(* PLC project SixAxisBoxPicker_Task.project, CODESYS CODESYS V3.5 SP16 Patch 4 for Safety V1.6.1 *)
(* stored: creationDateTime 2022-02-01T19:12:31.3073643, modificationDateTime 2022-02-01T19:06:40.3294124 *)

{attribute 'qualified_only'}
{attribute 'strict'}
{attribute 'to_string'}
TYPE
  E_mcMotionFbType :
  (
    moveCrcAbs := 0,
    moveCrcRel,
    moveDirAbs,
    moveDirRel,
    moveLinAbs,
    moveLinRel,
    // enums have to begin from zero and be sequential for this to work
    TotalNumberOfEnums
  );
END_TYPE

TYPE
  ST_haltParams :
  STRUCT
    lrDec     : LREAL;
    lrJrk     : LREAL;
    lrAccFctr : LREAL                         := 1;
    lrJrkFctr : LREAL                         := 1;
    smcCrdSys : SM3_Robotics.SMC_COORD_SYSTEM := SM3_Robotics.SMC_COORD_SYSTEM.ACS; // for logging halted position
  END_STRUCT
END_TYPE

TYPE
  ST_mcMoveParams :
  STRUCT
    eMcMotionFbType : E_mcMotionFbType;
    stMoveDirParams : ST_moveDirParams;
    stMoveCrcParams : ST_moveCrcParams;
    stMoveLinParams : ST_moveLinParams;
  END_STRUCT
END_TYPE

TYPE
  ST_moveCrcParams :
  STRUCT
    smcCrcMod       : SM3_Robotics.SMC_CIRC_MODE;
    smcPosRef_auxPt : SM3_Robotics.SMC_POS_REF;
    smcPosRef_endPt : SM3_Robotics.SMC_POS_REF;
    mcCrcPathChoice : SM3_Robotics.MC_CIRC_PATHCHOICE;
    lrVel           : LREAL;
    lrAcc           : LREAL;
    lrDec           : LREAL;
    lrJrk           : LREAL;
    smcCrdSys       : SM3_Robotics.SMC_COORD_SYSTEM;
    mcBufMode       : SM3_Common.MC_BUFFER_MODE       := SM3_Common.MC_BUFFER_MODE.Aborting;
    mcTrnMode       : SM3_Robotics.MC_TRANSITION_MODE := SM3_Robotics.MC_TRANSITION_MODE.TMNone;
    arrTrnPrm       : ARRAY[0..(SMC_RCNST.MAX_TRANS_PARAMS - 1)] OF LREAL;
    smcOrnMod       : SM3_Robotics.SMC_ORIENTATION_MODE;
    lrVelFctr       : LREAL := 1;
    lrAccFctr       : LREAL := 1;
    lrJrkFctr       : LREAL := 1;
  END_STRUCT
END_TYPE

TYPE
  ST_moveDirParams :
  STRUCT
    smcPosRef : SM3_Robotics.SMC_POS_REF;
    smcPtpTyp : SM3_Robotics.SMC_PTP_MOVEMENT_TYPE;
    smcCrdSys : SM3_Robotics.SMC_COORD_SYSTEM;
    mcBufMode : SM3_Common.MC_BUFFER_MODE       := SM3_Common.MC_BUFFER_MODE.Aborting;
    mcTrnMode : SM3_Robotics.MC_TRANSITION_MODE := SM3_Robotics.MC_TRANSITION_MODE.TMNone;
    arrTrnPrm : ARRAY[0..(SMC_RCNST.MAX_TRANS_PARAMS - 1)] OF LREAL;
    lrVelFctr : LREAL := 1;
    lrAccFctr : LREAL := 1;
    lrJrkFctr : LREAL := 1;
  END_STRUCT
END_TYPE

TYPE
  ST_moveLinParams :
  STRUCT
    smcPosRef : SM3_Robotics.SMC_POS_REF;
    lrVel     : LREAL;
    lrAcc     : LREAL;
    lrDec     : LREAL;
    lrJrk     : LREAL;
    smcCrdSys : SM3_Robotics.SMC_COORD_SYSTEM;
    mcBufMode : SM3_Common.MC_BUFFER_MODE       := SM3_Common.MC_BUFFER_MODE.Aborting;
    mcTrnMode : SM3_Robotics.MC_TRANSITION_MODE := SM3_Robotics.MC_TRANSITION_MODE.TMNone;
    arrTrnPrm : ARRAY[0..(SMC_RCNST.MAX_TRANS_PARAMS - 1)] OF LREAL;
    smcOrnMod : SM3_Robotics.SMC_ORIENTATION_MODE;
    lrVelFctr : LREAL := 1;
    lrAccFctr : LREAL := 1;
    lrJrkFctr : LREAL := 1;
  END_STRUCT
END_TYPE

TYPE
  ST_methConfig :
  STRUCT
    xGroupPowerOff : BOOL;
    xGroupPowerOn  : BOOL;
    xGroupEnable   : BOOL;
    xGroupDisable  : BOOL;
    xGroupHalt     : BOOL;
    xMoveCrcAbs    : BOOL;
    xMoveDirAbs    : BOOL;
    xCloseGripper  : BOOL;
    xOpenGripper   : BOOL;
  END_STRUCT
END_TYPE

TYPE
  T_MaxString : STRING(1000);
END_TYPE

(* global variable list GVL_Diag *)
VAR_GLOBAL
	
	//-------------------
	// EtherCAT diagnosis
	//-------------------
	ECDiag : FB_ECDiag;	// Instance of Ethercat Diagnosis

	MyECSlaves : stECSlaves := // Input Values for EtherCAT Diagnosis 		
		(
			uiNoSlaves := 10,
			arMyProductID := 
			[
			16#0002CF2F,	// FIO_Buskoppler_16DI_16DO	
			16#0002D7A8,  	// Safety PLC
			16#0002ECAD,  	// Kuhnke_FIO_Safety_SDI16_SDO4_1
			16#0002ECAD,  	// Kuhnke_FIO_Safety_SDI16_SDO4_2
			16#00000201, 	// Synapticon Somanet
			16#00000201, 	// Synapticon Somanet
			16#00000201, 	// Synapticon Somanet
			16#00000201, 	// Synapticon Somanet
			16#00000201, 	// Synapticon Somanet
			16#00000201 	// Synapticon Somanet
			]
		);	

	//-------------------
	// Motion diagnosis
	//-------------------
	AxisDiag : FB_AxisDiag;// Instance of Axis Diagnosis

	MyAxis : stAxis := 		// Input Values for Axis Diagnosis 
		(
		uiNoAxis := INT_TO_UINT(iNoConfigAxis),		// Number of Axis in project	
		arMyAxis :=			// Pointer to Axis 
			[
			ADR(A1),
			ADR(A2),
			ADR(A3),
			ADR(A4)
			]
		);
	
	//-------------------
	// Group diagnosis
	//-------------------
	GroupDiag : FB_GroupDiag;// Instance of Group Diagnosis

	//-------------------
	// Safety diagnosis
	//-------------------
	SafetyIODiag1 : FB_SafetyIODiag;// Instance of SafetyIO Diagnosis
	SafetyIODiag2 : FB_SafetyIODiag;// Instance of SafetyIO Diagnosis
	
	//-------------------
	// Task diagnosis
	//-------------------
	TaskDiag : FB_TaskDiag ; // Instance of Task Diagnosis
	MyTask : stTask := 		// Input Values for Task Diagnosis 
		(
			sAppName := 'Application',
			Watchdog :=
			[
				(Active := TRUE,WDTime:= 4000,Sensitivity:=2),  // Watchdog EtherCAT Task 1
				(Active := TRUE,WDTime:= 20000,Sensitivity:=2), // Watchdog Planning Task 2
				(Active := FALSE)								// Watchdog Settings Task 3
			]			
		);

END_VAR

INTERFACE I_machineState
METHOD METH_grpPwrOn
END_METHOD
METHOD METH_grpPwrOff
END_METHOD
METHOD METH_openGripper
END_METHOD
METHOD METH_groupHalt
VAR_INPUT
  stHaltParams : ST_haltParams;
END_VAR
VAR_OUTPUT
  xHaltFinished : BOOL;
END_VAR
END_METHOD
METHOD METH_closeGripper
END_METHOD
METHOD METH_moveToPosition
VAR_IN_OUT
  mcMoveLinkedList : COL.LinkedList;
END_VAR
VAR_OUTPUT
  xMotionFinished : BOOL;
END_VAR
END_METHOD
METHOD METH_groupEnable
END_METHOD
METHOD METH_groupDisable
END_METHOD
END_INTERFACE

INTERFACE I_mcMoveElement EXTENDS COL.IElement
METHOD METH_executeMcMove
VAR_IN_OUT
  axisGrpRefSm3 : SM3_Robotics.AXIS_GROUP_REF_SM3;
END_VAR
VAR_OUTPUT
  xDone        : BOOL;
  xBusy        : BOOL;
  xActive      : BOOL;
  xCmdAborted  : BOOL;
  xCmdAccepted : BOOL;
  xError       : BOOL;
  smcError     : SM3_Error.SMC_ERROR;
  smcMvmtId    : SM3_Common.SMC_Movement_Id;
END_VAR
END_METHOD
METHOD METH_resetMcMove
VAR_IN_OUT
  axisGrpRefSm3 : SM3_Robotics.AXIS_GROUP_REF_SM3;
END_VAR
END_METHOD
METHOD METH_setMcMoveParams
VAR_INPUT
  stMcMoveParams : ST_mcMoveParams;
  uliMotionIndx  : ULINT;
END_VAR
END_METHOD
PROPERTY INTERNAL PROP_mcMoveCrcAbs : SM3_Robotics.MC_MoveCircularAbsolute
END_PROPERTY
PROPERTY INTERNAL PROP_mcMoveCrcRel : SM3_Robotics.MC_MoveCircularRelative
END_PROPERTY
PROPERTY PROP_motionIndx : ULINT
END_PROPERTY
PROPERTY PROP_stMcMoveParams : ST_mcMoveParams
END_PROPERTY
PROPERTY INTERNAL PROP_mcMoveDirAbs : SM3_Robotics.MC_MoveDirectAbsolute
END_PROPERTY
PROPERTY INTERNAL PROP_mcMoveDirRel : SM3_Robotics.MC_MoveDirectRelative
END_PROPERTY
PROPERTY INTERNAL PROP_mcMoveLinAbs : SM3_Robotics.MC_MoveLinearAbsolute
END_PROPERTY
PROPERTY INTERNAL PROP_mcMoveLinRel : SM3_Robotics.MC_MoveLinearRelative
END_PROPERTY
END_INTERFACE

TYPE U_lrealToRawLintBits : UNION
  lrVal : LREAL;
  liVal : LINT;
END_UNION;
END_TYPE

FUNCTION F_getCommaDelimitedName : STRING
VAR_IN_OUT
  sCommaDelimitedNames : STRING; // comma delimited string
END_VAR
VAR
  sComma    : STRING := ',';
  iSplitPos : INT;

  fbLogAdd : FB_logAdd(pCmpName:=ADR(__POUNAME()));
END_VAR

            IF Standard.LEN(sCommaDelimitedNames) > 0 THEN
  // returns zero if comma not found
  iSplitPos := Standard.FIND(sCommaDelimitedNames, sComma);

  // copy string and set position to last character if comma not found
  IF iSplitPos = 0 THEN
    F_getCommaDelimitedName := sCommaDelimitedNames;
    iSplitPos := Standard.LEN(sCommaDelimitedNames);
  ELSE
    // extract name without comma
    F_getCommaDelimitedName := Standard.LEFT(sCommaDelimitedNames, (iSplitPos - 1));
  END_IF

  // delete name including comma
  sCommaDelimitedNames := Standard.DELETE(sCommaDelimitedNames, iSplitPos, 1);
ELSE
  fbLogAdd.METH_appendLog('Axis names string empty! Was it comma delimited? Were there too few axis names?');
  fbLogAdd.METH_printAppendedLogs();
  F_getCommaDelimitedName := '$00';
END_IF

          
END_FUNCTION

FUNCTION_BLOCK FB_logAdd
VAR
  sCmpName : STRING;
  sCurrLog : T_MaxString;

  // to check for duplicate states or log messages
  sPrevName : STRING      := '$00';
  sPrevLog  : T_MaxString := '$00';

  // for use as delimiter
  sNewline : STRING := '$0A';

  // does not need to be set beforehand as only used internally
  udiInternalCmpId : UDINT;
END_VAR

            
          

METHOD METH_appendLog
VAR_INPUT
  sLog     : T_MaxString;
  xNewline : BOOL := FALSE;
END_VAR
VAR
  sErrLog : STRING;
END_VAR
                  TM.Stu.StrConcatA(pstFrom:=ADR(sLog),
                  pstTo:=ADR(sCurrLog),
                  iBufferSize:=UINT_TO_INT(SIZEOF(sCurrLog)));

IF xNewline THEN
  TM.Stu.StrConcatA(pstFrom:=ADR(sNewline),
                    pstTo:=ADR(sCurrLog),
                    iBufferSize:=UINT_TO_INT(SIZEOF(sCurrLog)));
END_IF

IF TM.Stu.StrLenA(ADR(sCurrLog)) = (SIZEOF(sCurrLog) - 1) THEN
  sErrLog := Standard.CONCAT('SIZEOF(sCurrLog) = ', UINT_TO_STRING(SIZEOF(sCurrLog)));
  sErrLog := Standard.CONCAT(sErrLog, ' but it is not large enough for logger!');

  METH_printError(sErrLog);
END_IF

                
END_METHOD

METHOD METH_printAppendedLogs
VAR_INPUT
  sCmpName      : STRING := '$00';
  udiCmpVer     : UDINT  := 16#1;
  udiLogClass   : UDINT  := SM3_Basic.CmpLog.LogClass.LOG_USER_NOTIFY;
  udiErrorClass : UDINT  := SM3_Basic.Errors.ERR_FAILED;
END_VAR
VAR
  iSplitPos : INT         := 0;
  sSplitLog : STRING(255) := '$00';
END_VAR
                  // use persistent variable if not provided otherwise replace persistent one
IF sCmpName = '$00' THEN
  sCmpName := THIS^.sCmpName;
ELSE
  THIS^.sCmpName := sCmpName;
END_IF

// print log only if either state (set to sCmpName) or log message is different
// StrCmpA returns zero if strings are equal
IF TM.Stu.StrCmpA(ADR(sPrevLog), ADR(sCurrLog)) <> 0 OR
   TM.Stu.StrCmpA(ADR(sPrevName), ADR(sCmpName)) <> 0 THEN

  // store component name and log content to prevent lots of duplicates
  sPrevName := sCmpName;
  sPrevLog := sCurrLog;

  // set metadata i.e. component name, version etc.
  SM3_Basic.Component_Manager.CMAddComponent2(pszComponent:=sCmpName,
                                              udiVersion:=udiCmpVer,
                                              udiCmpId:=ADR(udiInternalCmpId),
                                              pResult:=0);

  SM3_Basic.CmpLog.LogAdd2(hLogger:=SM3_Basic.CmpLog.LOG_STD_LOGGER,
                           udiCmpID:=udiInternalCmpId,
                           udiClassID:=udiLogClass,
                           udiErrorID:=udiErrorClass,
                           udiInfoID:=1,
                           pszInfo:='(*--------------------------------------------------*)');

  // limit for pszComponent is 29 chars (will become *** if longer)
  IF Standard.LEN(sCmpName) > 29 THEN
    // so print sCmpName before actual log
    sCmpName := Standard.CONCAT('Cmp=', sCmpName);
    SM3_Basic.CmpLog.LogAdd2(hLogger:=SM3_Basic.CmpLog.LOG_STD_LOGGER,
                             udiCmpID:=udiInternalCmpId,
                             udiClassID:=udiLogClass,
                             udiErrorID:=udiErrorClass,
                             udiInfoID:=1,
                             pszInfo:=sCmpName);
  END_IF

  // split string using newline as delimiter
  WHILE TM.Stu.StrLenA(ADR(sCurrLog)) > 0 DO
    // StrFindA returns zero if substring at pst2 not found
    iSplitPos := TM.Stu.StrFindA(pst1:=ADR(sCurrLog),
                                 pst2:=ADR(sNewline),
                                 uiSearchStart:=1);

    // copy string and set position to last character if newline not found
    IF iSplitPos = 0 THEN
      sSplitLog := sCurrLog;
      iSplitPos := DINT_TO_INT(TM.Stu.StrLenA(ADR(sCurrLog)));
    ELSE
      // extract string without newline
      TM.Stu.StrMidA(pst:=ADR(sCurrLog),
                     uiInputBufferSize:=SIZEOF(sCurrLog),
                     iLength:=(iSplitPos - 1), // do not include newline
                     iPosition:=1,
                     pstResult:=ADR(sSplitLog),
                     uiResultBufferSize:=SIZEOF(sSplitLog));
    END_IF

    // delete extracted string and its corresponding newline from original
    TM.Stu.StrDeleteA(pby:=ADR(sCurrLog),
                      iLength:=iSplitPos, // include newline
                      iPosition:=1);

    // print extracted string with logger
    SM3_Basic.CmpLog.LogAdd2(hLogger:=SM3_Basic.CmpLog.LOG_STD_LOGGER,
                             udiCmpID:=udiInternalCmpId,
                             udiClassID:=udiLogClass,
                             udiErrorID:=udiErrorClass,
                             udiInfoID:=1,
                             pszInfo:=sSplitLog);
  END_WHILE
END_IF

// printing should flush buffer so delete anything remaining
TM.Stu.StrDeleteA(pby:=ADR(sCurrLog),
                  iLength:=DINT_TO_INT(TM.Stu.StrLenA(ADR(sCurrLog))),
                  iPosition:=1);

                
END_METHOD

//FB_Init is always available implicitly and it is used primarily for initialization.
//The return value is not evaluated. For a specific influence, you can also declare the
//methods explicitly and provide additional code there with the standard initialization
//code. You can evaluate the return value.
METHOD FB_Init : BOOL
VAR_INPUT
  bInitRetains : BOOL; // TRUE: the retain variables are initialized (reset warm / reset cold)
  bInCopyCode  : BOOL; // TRUE: the instance will be copied to the copy code afterward (online change) 
  pCmpName     : POINTER TO STRING;
END_VAR
                  // check if pointer is initialized before assigning
IF pCmpName <> 0 THEN
  THIS^.sCmpName := pCmpName^;
END_IF

                
END_METHOD

METHOD METH_appendTargetPositionLogs
VAR_INPUT
  smcCrdSys       : SM3_Robotics.SMC_COORD_SYSTEM;
  sAxisNames      : STRING; // comma delimited string
  smcPosRef       : SM3_Robotics.SMC_POS_REF;
  eMcMotionFbType : E_mcMotionFbType;
END_VAR
VAR
  diIndx : DINT;
END_VAR
                  IF smcCrdSys = SM3_Robotics.SMC_COORD_SYSTEM.ACS THEN
  METH_appendLog(sLog:='{');
  METH_appendLog(sLog:=sAxisNames);
  METH_appendLog(sLog:='}',
                 xNewline:=TRUE);
ELSE
  METH_appendLog(sLog:='{X,Y,Z,A,B,C}',
                 xNewline:=TRUE);
END_IF

METH_appendLog(sLog:='{');

FOR diIndx := LOWER_BOUND(smcPosRef.v, 1) TO UPPER_BOUND(smcPosRef.v, 1) BY 1 DO
  METH_appendLog(sLog:=LREAL_TO_STRING(smcPosRef.v[diIndx]));

  IF diIndx < UPPER_BOUND(smcPosRef.v, 1) THEN
    METH_appendLog(sLog:=',');
  END_IF
END_FOR

METH_appendLog(sLog:='}',
               xNewline:=TRUE);
							 
METH_appendLog(sLog:='with ');

METH_appendLog(sLog:=TO_STRING(eMcMotionFbType),
							 xNewline:=TRUE);

METH_appendLog(sLog:='in ');

CASE smcCrdSys OF
  SM3_Robotics.SMC_COORD_SYSTEM.ACS:
    METH_appendLog(sLog:='Axis Coordinate System',
                   xNewline:=TRUE);
  SM3_Robotics.SMC_COORD_SYSTEM.MCS:
    METH_appendLog(sLog:='Machine Coordinate System',
                   xNewline:=TRUE);
  SM3_Robotics.SMC_COORD_SYSTEM.PCS_1:
    METH_appendLog(sLog:='PCS_1',
                   xNewline:=TRUE);
  SM3_Robotics.SMC_COORD_SYSTEM.PCS_2:
    METH_appendLog(sLog:='PCS_2',
                   xNewline:=TRUE);
  SM3_Robotics.SMC_COORD_SYSTEM.TCS:
    METH_appendLog(sLog:='Tool Coordinate System',
                   xNewline:=TRUE);
  SM3_Robotics.SMC_COORD_SYSTEM.WCS:
    METH_appendLog(sLog:='World Coordinate System',
                   xNewline:=TRUE);
END_CASE

                
END_METHOD

METHOD METH_appendGrpStatusLog
VAR_IN_OUT
  axisGrpRefSm3 : SM3_Robotics.AXIS_GROUP_REF_SM3;
END_VAR
VAR_INPUT
  sGrpName : STRING;
END_VAR
VAR
  mcGrpReadStatus : SM3_Robotics.MC_GroupReadStatus;
END_VAR
                  mcGrpReadStatus(AxisGroup:=axisGrpRefSm3, Enable:=TRUE);

IF mcGrpReadStatus.Error THEN
  METH_printError(SM3_Error.SMC_ErrorString(ErrorID:=mcGrpReadStatus.ErrorID,
                                            Language:=SM3_Error.SMC_LANGUAGE_TYPE.english));

  RETURN;
END_IF

IF mcGrpReadStatus.Valid THEN
  METH_appendLog('Axis: ');
  METH_appendLog(sGrpName);
  METH_appendLog(' Status: ');

  IF mcGrpReadStatus.GroupDisabled THEN
    METH_appendLog('disabled');
  ELSIF mcGrpReadStatus.GroupStandby THEN
    METH_appendLog('standby');
  ELSIF mcGrpReadStatus.GroupMoving THEN
    METH_appendLog('moving');
  ELSIF mcGrpReadStatus.GroupHoming THEN
    METH_appendLog('homing');
  ELSIF mcGrpReadStatus.GroupStopping THEN
    METH_appendLog('stopping');
  ELSIF mcGrpReadStatus.GroupErrorStop THEN
    METH_appendLog('errorstop');
  END_IF

  // remember to add newline as used as delimiter by logger
  METH_appendLog(sNewline);
END_IF

                
END_METHOD

METHOD PRIVATE METH_printError
VAR_INPUT
  sErrLog : STRING;
END_VAR
VAR
  sTempLog  : T_MaxString;
  sTempName : STRING;
END_VAR
                  sTempLog := sCurrLog;
sTempName := sPrevName;

sCurrLog := sErrLog;
METH_printAppendedLogs(sCmpName:=__POUNAME());

sPrevName := sTempName;
sCurrLog := sTempLog;

                
END_METHOD

METHOD METH_appendStatusLogs
VAR_IN_OUT
  axisGrpRefSm3 : SM3_Robotics.AXIS_GROUP_REF_SM3;
END_VAR
VAR_INPUT
  sGrpName   : STRING;
  sAxisNames : STRING; // comma delimited string
END_VAR
VAR
  diIndx          : DINT;
  pAxisRefSm3     : POINTER TO SM3_Robotics.AXIS_REF_SM3;
END_VAR
                  IF axisGrpRefSm3.m_nNumAxes = 0 THEN
  METH_printError(Standard.CONCAT(sGrpName, ' has no axes!'));
  RETURN;
END_IF

FOR diIndx := LOWER_BOUND(axisGrpRefSm3.m_aAxes, 1) TO UPPER_BOUND(axisGrpRefSm3.m_aAxes, 1) BY 1 DO
  pAxisRefSm3 := axisGrpRefSm3.m_aAxes[diIndx].GetAxisRefPointer();
  METH_appendAxisStatusLog(axisRefSm3:=pAxisRefSm3^,
                           sAxisName:=F_getCommaDelimitedName(sAxisNames));
END_FOR

METH_appendGrpStatusLog(axisGrpRefSm3:=axisGrpRefSm3,
                        sGrpName:=sGrpName);

                
END_METHOD

METHOD METH_appendAxisStatusLog
VAR_IN_OUT
  axisRefSm3 : SM3_Basic.AXIS_REF_SM3;
END_VAR
VAR_INPUT
  sAxisName : STRING;
END_VAR
VAR
  mcReadStatus : SM3_Basic.MC_ReadStatus;
  mcReadActPos : SM3_Basic.MC_ReadActualPosition;
END_VAR
                  mcReadStatus(Axis:=axisRefSm3, Enable:=TRUE);

IF mcReadStatus.Error THEN
  METH_printError(SM3_Error.SMC_ErrorString(ErrorID:=mcReadStatus.ErrorID,
                                            Language:=SM3_Error.SMC_LANGUAGE_TYPE.english));

  RETURN;
END_IF

IF mcReadStatus.Valid THEN
  METH_appendLog('Axis: ');
  METH_appendLog(sAxisName);
  METH_appendLog(' Status: ');

  IF mcReadStatus.Disabled THEN
    METH_appendLog('disabled');
  ELSIF mcReadStatus.Errorstop THEN
    METH_appendLog('errorstop');
  ELSIF mcReadStatus.Stopping THEN
    METH_appendLog('stopping');
  ELSIF mcReadStatus.StandStill THEN
    METH_appendLog('standstill');
  ELSIF mcReadStatus.DiscreteMotion THEN
    METH_appendLog('discrete_motion');
  ELSIF mcReadStatus.ContinuousMotion THEN
    METH_appendLog('continuous_motion');
  ELSIF mcReadStatus.SynchronizedMotion THEN
    METH_appendLog('synchronized_motion');
  ELSIF mcReadStatus.Homing THEN
    METH_appendLog('homing');
  END_IF

  IF mcReadStatus.ConstantVelocity THEN
    METH_appendLog(' Speed: ConstantVelocity');
  ELSIF mcReadStatus.Accelerating THEN
    METH_appendLog(' Speed: Accelerating');
  ELSIF mcReadStatus.Decelerating THEN
    METH_appendLog(' Speed: Decelerating');
  END_IF

END_IF

mcReadActPos(Axis:=axisRefSm3,
             Enable:=TRUE);

IF mcReadActPos.Error THEN
  // remember to add newline as used as delimiter by logger
  METH_appendLog(sNewline);

  METH_printError(SM3_Error.SMC_ErrorString(ErrorID:=mcReadActPos.ErrorID,
                                            Language:=SM3_Error.SMC_LANGUAGE_TYPE.english));

  RETURN;
END_IF

IF mcReadActPos.Valid THEN
  METH_appendLog(' Position: ');
  METH_appendLog(LREAL_TO_STRING(mcReadActPos.Position));
END_IF

// remember to add newline as used as delimiter by logger
METH_appendLog(sNewline);

                
END_METHOD

METHOD METH_appendCurrentPositionLogs
VAR_IN_OUT
  axisGrpRefSm3 : SM3_Robotics.AXIS_GROUP_REF_SM3;
END_VAR
VAR_INPUT
  smcCrdSys  : SM3_Robotics.SMC_COORD_SYSTEM;
  sAxisNames : STRING; // comma delimted string
END_VAR
VAR
  mcGrpReadActPos : SM3_Robotics.MC_GroupReadActualPosition;
  diIndx          : DINT;
  sIndividualName : STRING;
  sCoordNames     : STRING := 'X,Y,Z,A,B,C';
END_VAR
                  mcGrpReadActPos(AxisGroup:=axisGrpRefSm3,
                Enable:=TRUE,
                CoordSystem:=smcCrdSys);

IF mcGrpReadActPos.Error THEN
  METH_printError(SM3_Error.SMC_ErrorString(ErrorID:=mcGrpReadActPos.ErrorID,
                                            Language:=SM3_Error.SMC_LANGUAGE_TYPE.english));

  RETURN;
END_IF

IF mcGrpReadActPos.Valid THEN
  METH_appendLog(sLog:='Current position:',
                 xNewline:=TRUE);

  FOR diIndx := LOWER_BOUND(mcGrpReadActPos.Position.v, 1) TO UPPER_BOUND(mcGrpReadActPos.Position.v, 1) BY 1 DO

    IF diIndx = LOWER_BOUND(mcGrpReadActPos.Position.v, 1) THEN
      METH_appendLog(sLog:='{ ');
    ELSE
      METH_appendLog(sLog:='  '); // blank space for better log alignment
    END_IF

    IF smcCrdSys = SM3_Robotics.SMC_COORD_SYSTEM.ACS THEN
      sIndividualName := F_getCommaDelimitedName(sAxisNames);
    ELSE
      sIndividualName := F_getCommaDelimitedName(sCoordNames);
    END_IF

    METH_appendLog(sLog:=sIndividualName);
		METH_appendLog(sLog:=': ');
    METH_appendLog(sLog:=LREAL_TO_STRING(mcGrpReadActPos.Position.v[diIndx]));

    IF diIndx = UPPER_BOUND(mcGrpReadActPos.Position.v, 1) THEN
      METH_appendLog(sLog:=' }',
                     xNewline:=TRUE);
    ELSE
      METH_appendLog(sLog:=',',
                     xNewline:=TRUE);
    END_IF
  END_FOR

END_IF

                
END_METHOD
END_FUNCTION_BLOCK

FUNCTION_BLOCK INTERNAL ABSTRACT FB_abstractEndMachineState EXTENDS FB_abstractMachineState IMPLEMENTS I_machineState

            sStateFb := __POUNAME();

          

METHOD METH_groupEnable
                  IF stMethConfig.xGroupEnable THEN
  METH_appendStateFbLog();
  METH_appendStatusLogs();
  METH_appendInfoLog('Enabling axes...');
  METH_printInfo(__POUNAME());

  pFbMachine^.METH_setState(pFbMachine^.PROP_enablingAxesState);
END_IF

                
END_METHOD

METHOD METH_grpPwrOn
                  IF stMethConfig.xGroupPowerOn THEN
  METH_appendStateFbLog();
  METH_appendStatusLogs();
  METH_appendInfoLog('Powering on axes...');
  METH_printInfo(__POUNAME());

  pFbMachine^.METH_setState(pFbMachine^.PROP_poweringOnState);
END_IF

                
END_METHOD

METHOD METH_grpPwrOff
                  IF stMethConfig.xGroupPowerOff THEN
  METH_appendStateFbLog();
  METH_appendStatusLogs();
  METH_appendInfoLog('Powering off axes...');
  METH_printInfo(__POUNAME());

  pFbMachine^.METH_setState(pFbMachine^.PROP_poweringOffState);
END_IF

                
END_METHOD

METHOD METH_openGripper
                  // IF stMethConfig.xOpenGripper THEN
// 	
// END_IF                           
                
END_METHOD

METHOD METH_groupHalt
VAR_INPUT
  stHaltParams : ST_haltParams;
END_VAR
VAR_OUTPUT
  xHaltFinished : BOOL;
END_VAR
                  // default values cannot be set in abstract or interface method
xHaltFinished := FALSE;

IF stMethConfig.xGroupHalt THEN
  METH_appendStateFbLog();
  METH_appendStatusLogs();
  METH_appendInfoLog('Halting axes...');
  METH_printInfo(__POUNAME());

  pFbMachine^.METH_setState(pFbMachine^.PROP_haltingState);
END_IF

                
END_METHOD

METHOD METH_closeGripper
                  // IF stMethConfig.xCloseGripper THEN
// END_IF                           
                
END_METHOD

METHOD METH_moveToPosition
VAR_IN_OUT
  mcMoveLinkedList : COL.LinkedList;
END_VAR
VAR_OUTPUT
  xMotionFinished : BOOL;
END_VAR
VAR
  linkedListIterator : COL.LinkedListIterator;
  itfLinkedListElem  : COL.IElement;
  itfMcMoveElement   : I_mcMoveElement;
  stMcMoveParams     : ST_mcMoveParams;

  mcMoveLinkedListInfo  : __SYSTEM.VAR_INFO;
  itfLinkedListElemInfo : __SYSTEM.VAR_INFO;
  itfMcMoveElementInfo  : __SYSTEM.VAR_INFO;
END_VAR
                  // default values cannot be set in abstract or interface method
xMotionFinished := FALSE;

IF stMethConfig.xMoveDirAbs THEN

  mcMoveLinkedListInfo := __VARINFO(mcMoveLinkedList);

  IF mcMoveLinkedList.CountElements() <= 0 THEN
    METH_appendInfoLog('No elements in ');
    METH_appendInfoLog(mcMoveLinkedListInfo.Symbol);
    METH_appendInfoLog('!');
  ELSE
    mcMoveLinkedList.ElementIterator(itfIterator:=linkedListIterator);

    WHILE linkedListIterator.HasNext() DO
      linkedListIterator.Next(itfElement=>itfLinkedListElem);

      itfLinkedListElemInfo := __VARINFO(itfLinkedListElem);
      itfMcMoveElementInfo := __VARINFO(itfMcMoveElement);

      IF NOT __QUERYINTERFACE(itfLinkedListElem, itfMcMoveElement) THEN
        METH_appendInfoLog('Unable to convert ');
        METH_appendInfoLog(itfLinkedListElemInfo.Symbol);
        METH_appendInfoLog(' to ');
        METH_appendInfoLog(itfMcMoveElementInfo.Symbol);
        METH_appendInfoLog('!');
      ELSE
        METH_appendStateFbLog();
        METH_appendStatusLogs();
        METH_appendInfoLog('Moving to position...');

        stMcMoveParams := itfMcMoveElement.PROP_stMcMoveParams;

        CASE stMcMoveParams.eMcMotionFbType OF

          E_mcMotionFbType.moveCrcAbs:
            METH_appendInfoLog('Not implemented yet!');

          E_mcMotionFbType.moveCrcRel:
            METH_appendInfoLog('Not implemented yet!');

          E_mcMotionFbType.moveDirAbs:
            METH_appendTargetPositionLogs(smcCrdSys:=stMcMoveParams.stMoveDirParams.smcCrdSys,
                                          smcPosRef:=stMcMoveParams.stMoveDirParams.smcPosRef,
                                          eMcMotionFbType:=stMcMoveParams.eMcMotionFbType);

          E_mcMotionFbType.moveDirRel:
            METH_appendTargetPositionLogs(smcCrdSys:=stMcMoveParams.stMoveDirParams.smcCrdSys,
                                          smcPosRef:=stMcMoveParams.stMoveDirParams.smcPosRef,
                                          eMcMotionFbType:=stMcMoveParams.eMcMotionFbType);

          E_mcMotionFbType.moveLinAbs:
            METH_appendTargetPositionLogs(smcCrdSys:=stMcMoveParams.stMoveLinParams.smcCrdSys,
                                          smcPosRef:=stMcMoveParams.stMoveLinParams.smcPosRef,
                                          eMcMotionFbType:=stMcMoveParams.eMcMotionFbType);

          E_mcMotionFbType.moveLinRel:
            METH_appendTargetPositionLogs(smcCrdSys:=stMcMoveParams.stMoveLinParams.smcCrdSys,
                                          smcPosRef:=stMcMoveParams.stMoveLinParams.smcPosRef,
                                          eMcMotionFbType:=stMcMoveParams.eMcMotionFbType);

        END_CASE

        METH_printInfo(__POUNAME());
      END_IF
    END_WHILE
  END_IF

  pFbMachine^.METH_setState(pFbMachine^.PROP_movingToPositionState);
END_IF

                
END_METHOD

METHOD METH_groupDisable
                  IF stMethConfig.xGroupDisable THEN
  METH_appendStateFbLog();
  METH_appendStatusLogs();
  METH_appendInfoLog('Disabling axes...');
  METH_printInfo(__POUNAME());

  pFbMachine^.METH_setState(pFbMachine^.PROP_disablingAxesState);
END_IF

                
END_METHOD
END_FUNCTION_BLOCK

FUNCTION_BLOCK INTERNAL FB_disabledAxesState EXTENDS FB_abstractEndMachineState

            sStateFb := __POUNAME();

stMethConfig.xGroupPowerOff := TRUE;
stMethConfig.xGroupPowerOn  := FALSE;
stMethConfig.xGroupEnable   := TRUE;
stMethConfig.xGroupDisable  := FALSE;
stMethConfig.xMoveDirAbs    := FALSE;
stMethConfig.xGroupHalt     := FALSE;
stMethConfig.xCloseGripper  := FALSE;
stMethConfig.xOpenGripper   := FALSE;

          
END_FUNCTION_BLOCK

FUNCTION_BLOCK INTERNAL FB_enabledAxesState EXTENDS FB_abstractEndMachineState

            sStateFb := __POUNAME();

stMethConfig.xGroupPowerOff := FALSE;
stMethConfig.xGroupPowerOn  := FALSE;
stMethConfig.xGroupEnable   := FALSE;
stMethConfig.xGroupDisable  := TRUE;
stMethConfig.xMoveDirAbs    := TRUE;
stMethConfig.xGroupHalt     := TRUE;
stMethConfig.xCloseGripper  := TRUE;
stMethConfig.xOpenGripper   := TRUE;

          
END_FUNCTION_BLOCK

FUNCTION_BLOCK INTERNAL FB_haltedState EXTENDS FB_abstractEndMachineState

            sStateFb := __POUNAME();

stMethConfig.xGroupPowerOff := FALSE;
stMethConfig.xGroupPowerOn  := FALSE;
stMethConfig.xGroupEnable   := FALSE;
stMethConfig.xGroupDisable  := TRUE;
stMethConfig.xMoveDirAbs    := TRUE;
stMethConfig.xGroupHalt     := TRUE;
stMethConfig.xCloseGripper  := TRUE;
stMethConfig.xOpenGripper   := TRUE;

          
END_FUNCTION_BLOCK

FUNCTION_BLOCK INTERNAL FB_movedToPositionState EXTENDS FB_abstractEndMachineState

            sStateFb := __POUNAME();

stMethConfig.xGroupPowerOff := FALSE;
stMethConfig.xGroupPowerOn  := FALSE;
stMethConfig.xGroupEnable   := FALSE;
stMethConfig.xGroupDisable  := TRUE;
stMethConfig.xMoveDirAbs    := TRUE;
stMethConfig.xGroupHalt     := TRUE;
stMethConfig.xCloseGripper  := TRUE;
stMethConfig.xOpenGripper   := TRUE;

          
END_FUNCTION_BLOCK

FUNCTION_BLOCK INTERNAL FB_poweredOffState EXTENDS FB_abstractEndMachineState

            sStateFb := __POUNAME();

stMethConfig.xGroupPowerOff := FALSE;
stMethConfig.xGroupPowerOn  := TRUE;
stMethConfig.xGroupEnable   := FALSE;
stMethConfig.xGroupDisable  := FALSE;
stMethConfig.xMoveDirAbs    := FALSE;
stMethConfig.xGroupHalt     := FALSE;
stMethConfig.xCloseGripper  := FALSE;
stMethConfig.xOpenGripper   := FALSE;

          
END_FUNCTION_BLOCK

FUNCTION_BLOCK INTERNAL FB_poweredOnState EXTENDS FB_abstractEndMachineState

            sStateFb := __POUNAME();

stMethConfig.xGroupPowerOff := TRUE;
stMethConfig.xGroupPowerOn  := FALSE;
stMethConfig.xGroupEnable   := TRUE;
stMethConfig.xGroupDisable  := FALSE;
stMethConfig.xMoveDirAbs    := FALSE;
stMethConfig.xGroupHalt     := FALSE;
stMethConfig.xCloseGripper  := FALSE;
stMethConfig.xOpenGripper   := FALSE;

          
END_FUNCTION_BLOCK

FUNCTION_BLOCK INTERNAL ABSTRACT FB_abstractMachineState
VAR
  pFbMachine   : POINTER TO FB_machine;
  pFbLogAdd    : POINTER TO FB_logAdd; // centralized in FB_machine
  sStateFb     : STRING;
  stMethConfig : ST_methConfig;
END_VAR

            sStateFb := __POUNAME();

          

//FB_Init is always available implicitly and it is used primarily for initialization.
//The return value is not evaluated. For a specific influence, you can also declare the
//methods explicitly and provide additional code there with the standard initialization
//code. You can evaluate the return value.
METHOD FB_Init : BOOL
VAR_INPUT
  bInitRetains : BOOL; // TRUE: the retain variables are initialized (reset warm / reset cold)
  bInCopyCode  : BOOL; // TRUE: the instance will be copied to the copy code afterward (online change)   
  pFbMachine   : POINTER TO FB_machine;
END_VAR
                  THIS^.pFbMachine := pFbMachine;
THIS^.pFbLogAdd := THIS^.pFbMachine^.PROP_fbLogAddPointer;

                
END_METHOD

METHOD PROTECTED METH_printInfo
VAR_INPUT
  sCmpName : STRING;
END_VAR
                  pFbLogAdd^.METH_printAppendedLogs(sCmpName:=sCmpName,
                                  udiErrorClass:=SM3_Basic.CmpLog.LogClass.LOG_INFO);

                
END_METHOD

METHOD PROTECTED METH_printSmcError
VAR_INPUT
  smcErrorId : SM3_Error.SMC_ERROR;
  sCmpName   : STRING;
END_VAR
                  pFbLogAdd^.METH_appendLog(sLog:=SM3_Error.SMC_ErrorString(ErrorID:=smcErrorId,
                                                          Language:=SM3_Error.SMC_LANGUAGE_TYPE.english));

pFbLogAdd^.METH_printAppendedLogs(sCmpName:=sCmpName);

                
END_METHOD

METHOD PROTECTED METH_appendStatusLogs
                  pFbLogAdd^.METH_appendStatusLogs(axisGrpRefSm3:=pFbMachine^.PROP_axisGroupPointer^,
                                 sGrpName:=pFbMachine^.sGrpName,
                                 sAxisNames:=pFbMachine^.sAxisNames);

                
END_METHOD

METHOD PROTECTED METH_appendInfoLog
VAR_INPUT
  sInfoMsg : STRING;
END_VAR
                  pFbLogAdd^.METH_appendLog(sLog:=sInfoMsg,
                          xNewline:=TRUE);

                
END_METHOD

METHOD PROTECTED METH_appendTargetPositionLogs
VAR_INPUT
  smcCrdSys : SM3_Robotics.SMC_COORD_SYSTEM;
  smcPosRef : SM3_Robotics.SMC_POS_REF;
	eMcMotionFbType : E_mcMotionFbType;
END_VAR
                  pFbLogAdd^.METH_appendTargetPositionLogs(smcCrdSys:=smcCrdSys,
                                         sAxisNames:=pFbMachine^.sAxisNames,
                                         smcPosRef:=smcPosRef,
                                         eMcMotionFbType:=eMcMotionFbType);

                
END_METHOD

METHOD PROTECTED METH_appendStateFbLog
                  pFbLogAdd^.METH_appendLog(sLog:='Current state: ');
pFbLogAdd^.METH_appendLog(sLog:=sStateFb,
                          xNewline:=TRUE);

                
END_METHOD

METHOD PROTECTED METH_appendCurrentPositionLogs
VAR_INPUT
  smcCrdSys : SM3_Robotics.SMC_COORD_SYSTEM;
END_VAR
                  pFbLogAdd^.METH_appendCurrentPositionLogs(axisGrpRefSm3:=pFbMachine^.PROP_axisGroupPointer^,
                                          sAxisNames:=pFbMachine^.sAxisNames,
                                          smcCrdSys:=smcCrdSys);

                
END_METHOD
END_FUNCTION_BLOCK

FUNCTION_BLOCK FB_machine
VAR
  // everything initialized in FB_Init
  rAxisGrpRefSm3 : REFERENCE TO SM3_Robotics.AXIS_GROUP_REF_SM3;
  sGrpName       : STRING;
  sAxisNames     : STRING; // comma delimited string

  // logger used by FB_baseMachineState
  fbLogAdd : FB_logAdd(pCmpName:=ADR(__POUNAME()));

  // state pattern
  itfMachineState : I_machineState := fbPoweredOff;

  // end states
  fbPoweredOff      : FB_poweredOffState(THIS);
  fbPoweredOn       : FB_poweredOnState(THIS);
  fbEnabledAxes     : FB_enabledAxesState(THIS);
  fbDisabledAxes    : FB_disabledAxesState(THIS);
  fbHalted          : FB_haltedState(THIS);
  fbMovedToPosition : FB_movedToPositionState(THIS);
  // interim states
  fbPoweringOff      : FB_poweringOffState(THIS);
  fbPoweringOn       : FB_poweringOnState(THIS);
  fbEnablingAxes     : FB_enablingAxesState(THIS);
  fbDisablingAxes    : FB_disablingAxesState(THIS);
  fbHalting          : FB_haltingState(THIS);
  fbMovingToPosition : FB_movingToPositionState(THIS);
END_VAR

            
          

METHOD INTERNAL METH_setState
VAR_INPUT
  itfNewState : I_machineState;
END_VAR
                  itfMachineState := itfNewState;

                
END_METHOD

METHOD METH_groupEnable
                  itfMachineState.METH_groupEnable();

                
END_METHOD

//FB_Init is always available implicitly and it is used primarily for initialization.
//The return value is not evaluated. For a specific influence, you can also declare the
//methods explicitly and provide additional code there with the standard initialization
//code. You can evaluate the return value.
METHOD FB_Init : BOOL
VAR_INPUT
  bInitRetains   : BOOL; // TRUE: the retain variables are initialized (reset warm / reset cold)
  bInCopyCode    : BOOL; // TRUE: the instance will be copied to the copy code afterward (online change)
  rAxisGrpRefSm3 : REFERENCE TO SM3_Robotics.AXIS_GROUP_REF_SM3;
  sGrpName       : STRING;
  sAxisNames     : STRING; // comma delimited string
END_VAR
                  IF __ISVALIDREF(rAxisGrpRefSm3) THEN
	THIS^.rAxisGrpRefSm3 REF= rAxisGrpRefSm3;
END_IF
THIS^.sGrpName := sGrpName;
THIS^.sAxisNames := sAxisNames;

// initialize respective ST_methConfig 
// end states
THIS^.fbPoweredOff();
THIS^.fbPoweredOn();
THIS^.fbEnabledAxes();
THIS^.fbDisabledAxes();
THIS^.fbHalted();
// THIS^.fbMovedCrcAbs();
THIS^.fbMovedToPosition();
// interim states
THIS^.fbPoweringOff();
THIS^.fbPoweringOn();
THIS^.fbEnablingAxes();
THIS^.fbDisablingAxes();
THIS^.fbHalting();
// THIS^.fbMovingCrcAbs();
THIS^.fbMovingToPosition();

                
END_METHOD

METHOD METH_groupDisable
                  itfMachineState.METH_groupDisable();

                
END_METHOD

METHOD METH_grpPwrOn
                  itfMachineState.METH_grpPwrOn();

                
END_METHOD

METHOD METH_grpPwrOff
                  itfMachineState.METH_grpPwrOff();

                
END_METHOD

METHOD METH_moveToPosition
VAR_IN_OUT
  mcMoveLinkedList : COL.LinkedList;
END_VAR
VAR_OUTPUT
  xMotionFinished : BOOL;
END_VAR
                  itfMachineState.METH_moveToPosition(mcMoveLinkedList,
                                    xMotionFinished=>xMotionFinished);

                
END_METHOD

METHOD METH_groupHalt
VAR_INPUT
  stHaltParams : ST_haltParams;
END_VAR
VAR_OUTPUT
  xHaltFinished : BOOL;
END_VAR
                  itfMachineState.METH_groupHalt(stHaltParams:=stHaltParams,
                          xHaltFinished=>xHaltFinished);

                
END_METHOD

PROPERTY INTERNAL PROP_poweringOnState : I_machineState
GET
                    PROP_poweringOnState := fbPoweringOn;

                  
END_GET
END_PROPERTY

PROPERTY INTERNAL PROP_poweredOnState : I_machineState
GET
                    PROP_poweredOnState := fbPoweredOn;

                  
END_GET
END_PROPERTY

PROPERTY INTERNAL PROP_poweredOffState : I_machineState
GET
                    PROP_poweredOffState := fbPoweredOff;

                  
END_GET
END_PROPERTY

PROPERTY INTERNAL PROP_fbLogAddPointer : POINTER TO FB_logAdd
GET
                    PROP_fbLogAddPointer := ADR(fbLogAdd);

                  
END_GET
END_PROPERTY

PROPERTY PROP_axisGroupPointer : POINTER TO AXIS_GROUP_REF_SM3
GET
                    PROP_axisGroupPointer := ADR(rAxisGrpRefSm3);

                  
END_GET
END_PROPERTY

PROPERTY INTERNAL PROP_poweringOffState : I_machineState
GET
                    PROP_poweringOffState := fbPoweringOff;

                  
END_GET
END_PROPERTY

PROPERTY INTERNAL PROP_enabledAxesState : I_machineState
GET
                    PROP_enabledAxesState := fbEnabledAxes;

                  
END_GET
END_PROPERTY

PROPERTY INTERNAL PROP_enablingAxesState : I_machineState
GET
                    PROP_enablingAxesState := fbEnablingAxes;

                  
END_GET
END_PROPERTY

PROPERTY INTERNAL PROP_disabledAxesState : I_machineState
GET
                    PROP_disabledAxesState := fbDisabledAxes;

                  
END_GET
END_PROPERTY

PROPERTY INTERNAL PROP_disablingAxesState : I_machineState
GET
                    PROP_disablingAxesState := fbDisablingAxes;

                  
END_GET
END_PROPERTY

PROPERTY INTERNAL PROP_movedToPositionState : I_machineState
GET
                    PROP_movedToPositionState := fbMovedToPosition;

                  
END_GET
END_PROPERTY

PROPERTY INTERNAL PROP_movingToPositionState : I_machineState
GET
                    PROP_movingToPositionState := fbMovingToPosition;

                  
END_GET
END_PROPERTY

PROPERTY INTERNAL PROP_haltingState : I_machineState
GET
                    PROP_haltingState := fbHalting;

                  
END_GET
END_PROPERTY

PROPERTY INTERNAL PROP_haltedState : I_machineState
GET
                    PROP_haltedState := fbHalted;

                  
END_GET
END_PROPERTY
END_FUNCTION_BLOCK

FUNCTION_BLOCK INTERNAL ABSTRACT FB_abstractInterimMachineState EXTENDS FB_abstractMachineState IMPLEMENTS I_machineState

            sStateFb := __POUNAME();

          

METHOD METH_groupEnable
VAR
  mcGrpEnable : SM3_Robotics.MC_GroupEnable;
END_VAR
                  IF stMethConfig.xGroupEnable THEN
  mcGrpEnable(AxisGroup:=pFbMachine^.PROP_axisGroupPointer^,
              Execute:=TRUE);

  IF mcGrpEnable.Error THEN
    METH_printSmcError(smcErrorId:=mcGrpEnable.ErrorID,
                    sCmpName:=__POUNAME());

    RETURN;
  END_IF

  METH_appendStateFbLog();
  METH_appendStatusLogs();

  IF mcGrpEnable.Done THEN
    METH_appendInfoLog('Enabled axes');

    pFbMachine^.METH_setState(pFbMachine^.PROP_enabledAxesState);
  ELSE
    pFbMachine^.METH_setState(pFbMachine^.PROP_enablingAxesState);
  END_IF

  METH_printInfo(__POUNAME());

END_IF

                
END_METHOD

METHOD METH_openGripper
                  // IF stMethConfig.xOpenGripper THEN
// 	
// END_IF                             
                
END_METHOD

METHOD METH_groupHalt
VAR_INPUT
  stHaltParams : ST_haltParams;
END_VAR
VAR_OUTPUT
  xHaltFinished : BOOL;
END_VAR
VAR
  mcGrpHalt    : SM3_Robotics.MC_GroupHalt;
END_VAR
                  // default values cannot be set in abstract or interface method
xHaltFinished := FALSE;

IF stMethConfig.xGroupHalt THEN

  mcGrpHalt(AxisGroup:=pFbMachine^.PROP_axisGroupPointer^,
            Execute:=TRUE,
            Deceleration:=stHaltParams.lrDec,
            Jerk:=stHaltParams.lrJrk,
            AccFactor:=stHaltParams.lrAccFctr,
            JerkFactor:=stHaltParams.lrJrkFctr);

  IF mcGrpHalt.Error THEN
    METH_printSmcError(smcErrorId:=mcGrpHalt.ErrorID,
                    sCmpName:=__POUNAME());

    RETURN;
  END_IF

  METH_appendStateFbLog();
  METH_appendStatusLogs();

  IF mcGrpHalt.Done THEN
    METH_appendInfoLog('Halted');

    // remember to reset execute since persistent FB otherwise will not move to next position when called
    mcGrpHalt(AxisGroup:=pFbMachine^.PROP_axisGroupPointer^,
              Execute:=FALSE);

    xHaltFinished := TRUE;

    pFbMachine^.METH_setState(pFbMachine^.PROP_haltedState);
  ELSE
    pFbMachine^.METH_setState(pFbMachine^.PROP_haltingState);
  END_IF

  // axis positions already printed in METH_appendStatusLogs()
  IF stHaltParams.smcCrdSys <> SM3_Robotics.SMC_COORD_SYSTEM.ACS THEN
    METH_appendCurrentPositionLogs(smcCrdSys:=stHaltParams.smcCrdSys);
  END_IF

  METH_printInfo(__POUNAME());

END_IF

                
END_METHOD

METHOD METH_grpPwrOff
VAR
  smcGrpPwr : SM3_Robotics.SMC_GroupPower;
END_VAR
                  IF stMethConfig.xGroupPowerOff THEN
  smcGrpPwr(AxisGroup:=pFbMachine^.PROP_axisGroupPointer^,
            Enable:=TRUE,
            bRegulatorOn:=FALSE,
            bDriveStart:=FALSE);

  IF smcGrpPwr.Error THEN
    METH_printSmcError(smcErrorId:=smcGrpPwr.ErrorID,
                    sCmpName:=__POUNAME());

    RETURN;
  END_IF

  METH_appendStateFbLog();
  METH_appendStatusLogs();

  IF smcGrpPwr.Status THEN
    METH_appendInfoLog('Powered off axes');

    pFbMachine^.METH_setState(pFbMachine^.PROP_poweredOffState);
  ELSE
    pFbMachine^.METH_setState(pfbmachine^.PROP_poweringOffState);
  END_IF

  METH_printInfo(__POUNAME());

END_IF

                
END_METHOD

METHOD METH_grpPwrOn
VAR
  smcGrpPwr : SM3_Robotics.SMC_GroupPower;
END_VAR
                  IF stMethConfig.xGroupPowerOn THEN
  smcGrpPwr(AxisGroup:=pFbMachine^.PROP_axisGroupPointer^,
            Enable:=TRUE,
            bRegulatorOn:=TRUE,
            bDriveStart:=TRUE);

  IF smcGrpPwr.Error THEN
    METH_printSmcError(smcErrorId:=smcGrpPwr.ErrorID,
                    sCmpName:=__POUNAME());

    RETURN;
  END_IF

  METH_appendStateFbLog();
  METH_appendStatusLogs();

  IF smcGrpPwr.Status THEN
    METH_appendInfoLog('Powered on axes');

    pFbMachine^.METH_setState(pFbMachine^.PROP_poweredOnState);
  ELSE
    pFbMachine^.METH_setState(pfbmachine^.PROP_poweringOnState);
  END_IF

  METH_printInfo(__POUNAME());

END_IF

                
END_METHOD

METHOD METH_closeGripper
                  // IF stMethConfig.xCloseGripper THEN
// 	
// END_IF                             
                
END_METHOD

METHOD METH_moveToPosition
VAR_IN_OUT
  mcMoveLinkedList : COL.LinkedList;
END_VAR
VAR_OUTPUT
  xMotionFinished : BOOL;
END_VAR
VAR
	linkedListIterator : COL.LinkedListIterator;
  itfLinkedListElem  : COL.IElement;
  itfMcMoveElement   : I_mcMoveElement;
  stMcMoveParams     : ST_mcMoveParams;

  mcMoveLinkedListInfo  : __SYSTEM.VAR_INFO;
  itfLinkedListElemInfo : __SYSTEM.VAR_INFO;
  itfMcMoveElementInfo  : __SYSTEM.VAR_INFO;

  xDone        : BOOL;
  xBusy        : BOOL;
  xActive      : BOOL;
  xCmdAborted  : BOOL;
  xCmdAccepted : BOOL;
  xError       : BOOL;
  smcError     : SM3_Error.SMC_ERROR;
  smcMvmtId    : SM3_Common.SMC_Movement_Id;
END_VAR
                  // default values cannot be set in abstract or interface method
xMotionFinished := FALSE;

IF stMethConfig.xMoveDirAbs THEN

  mcMoveLinkedListInfo := __VARINFO(mcMoveLinkedList);

  IF mcMoveLinkedList.CountElements() <= 0 THEN
    METH_appendInfoLog('No elements in ');
    METH_appendInfoLog(mcMoveLinkedListInfo.Symbol);
    METH_appendInfoLog('!');
  ELSE
    mcMoveLinkedList.ElementIterator(itfIterator:=linkedListIterator);

    WHILE linkedListIterator.HasNext() DO
      linkedListIterator.Next(itfElement=>itfLinkedListElem);

      itfLinkedListElemInfo := __VARINFO(itfLinkedListElem);
      itfMcMoveElementInfo := __VARINFO(itfMcMoveElement);

      IF NOT __QUERYINTERFACE(itfLinkedListElem, itfMcMoveElement) THEN
        METH_appendInfoLog('Unable to convert ');
        METH_appendInfoLog(itfLinkedListElemInfo.Symbol);
        METH_appendInfoLog(' to ');
        METH_appendInfoLog(itfMcMoveElementInfo.Symbol);
        METH_appendInfoLog('!');
      ELSE
        itfMcMoveElement.METH_executeMcMove(axisGrpRefSm3:=pFbMachine^.PROP_axisGroupPointer^,
                                            xDone=>xDone,
                                            xBusy=>xBusy,
                                            xActive=>xActive,
                                            xCmdAborted=>xCmdAborted,
                                            xCmdAccepted=>xCmdAccepted,
                                            xError=>xError,
                                            smcError=>smcError,
                                            smcMvmtId=>smcMvmtId);

        IF xError THEN
          METH_printSmcError(smcErrorId:=smcError,
                             sCmpName:=__POUNAME());

          RETURN;
        END_IF

        METH_appendStateFbLog();
        METH_appendStatusLogs();

        stMcMoveParams := itfMcMoveElement.PROP_stMcMoveParams;

        IF xDone THEN
          METH_appendInfoLog('Moved to position');

          // need to implement method containing case statement for appendTargetPositionLogs
          METH_appendTargetPositionLogs(smcCrdSys:=stMcMoveParams.stMoveDirParams.smcCrdSys,
                                        smcPosRef:=stMcMoveParams.stMoveDirParams.smcPosRef,
                                        eMcMotionFbType:=E_mcMotionFbType.moveDirAbs);

          // remember to reset execute since persistent FB otherwise will not move to next position when called
          itfMcMoveElement.METH_resetMcMove(pFbMachine^.PROP_axisGroupPointer^);

          xMotionFinished := TRUE;

          pFbMachine^.METH_setState(pFbMachine^.PROP_movedToPositionState);
        ELSE
          // axis positions already printed in METH_appendStatusLogs()
          IF stMcMoveParams.stMoveDirParams.smcCrdSys <> SM3_Robotics.SMC_COORD_SYSTEM.ACS THEN
            METH_appendCurrentPositionLogs(smcCrdSys:=stMcMoveParams.stMoveDirParams.smcCrdSys);
          END_IF

          pFbMachine^.METH_setState(pFbMachine^.PROP_movingToPositionState);
        END_IF

      END_IF

      METH_printInfo(__POUNAME());
    END_WHILE
  END_IF
END_IF

                
END_METHOD

METHOD METH_groupDisable
VAR
  mcGrpDisable : SM3_Robotics.MC_GroupDisable;
END_VAR
                  IF stMethConfig.xGroupDisable THEN
  mcGrpDisable(AxisGroup:=pFbMachine^.PROP_axisGroupPointer^,
               Execute:=TRUE);

  IF mcGrpDisable.Error THEN
    METH_printSmcError(smcErrorId:=mcGrpDisable.ErrorID,
                    sCmpName:=__POUNAME());

    RETURN;
  END_IF

  METH_appendStateFbLog();
  METH_appendStatusLogs();

  IF mcGrpDisable.Done THEN
    METH_appendInfoLog('Disabled axes');

    pFbMachine^.METH_setState(pFbMachine^.PROP_disabledAxesState);
  ELSE
    pFbMachine^.METH_setState(pFbMachine^.PROP_disablingAxesState);
  END_IF

  METH_printInfo(__POUNAME());

END_IF

                
END_METHOD
END_FUNCTION_BLOCK

FUNCTION_BLOCK INTERNAL FB_disablingAxesState EXTENDS FB_abstractInterimMachineState

            sStateFb := __POUNAME();

stMethConfig.xGroupPowerOff := FALSE;
stMethConfig.xGroupPowerOn  := FALSE;
stMethConfig.xGroupEnable   := FALSE;
stMethConfig.xGroupDisable  := TRUE;
stMethConfig.xMoveDirAbs    := FALSE;
stMethConfig.xGroupHalt     := FALSE;
stMethConfig.xCloseGripper  := FALSE;
stMethConfig.xOpenGripper   := FALSE;

          
END_FUNCTION_BLOCK

FUNCTION_BLOCK INTERNAL FB_enablingAxesState EXTENDS FB_abstractInterimMachineState

            sStateFb := __POUNAME();

stMethConfig.xGroupPowerOff := FALSE;
stMethConfig.xGroupPowerOn  := FALSE;
stMethConfig.xGroupEnable   := TRUE;
stMethConfig.xGroupDisable  := FALSE;
stMethConfig.xMoveDirAbs    := FALSE;
stMethConfig.xGroupHalt     := FALSE;
stMethConfig.xCloseGripper  := FALSE;
stMethConfig.xOpenGripper   := FALSE;

          
END_FUNCTION_BLOCK

FUNCTION_BLOCK INTERNAL FB_haltingState EXTENDS FB_abstractInterimMachineState

            sStateFb := __POUNAME();

stMethConfig.xGroupPowerOff := FALSE;
stMethConfig.xGroupPowerOn  := FALSE;
stMethConfig.xGroupEnable   := FALSE;
stMethConfig.xGroupDisable  := FALSE;
stMethConfig.xMoveDirAbs    := FALSE;
stMethConfig.xGroupHalt     := TRUE;
stMethConfig.xCloseGripper  := FALSE;
stMethConfig.xOpenGripper   := FALSE;

          
END_FUNCTION_BLOCK

FUNCTION_BLOCK INTERNAL FB_movingToPositionState EXTENDS FB_abstractInterimMachineState

            sStateFb := __POUNAME();

stMethConfig.xGroupPowerOff := FALSE;
stMethConfig.xGroupPowerOn  := FALSE;
stMethConfig.xGroupEnable   := FALSE;
stMethConfig.xGroupDisable  := FALSE;
stMethConfig.xMoveDirAbs    := TRUE;
stMethConfig.xGroupHalt     := TRUE;
stMethConfig.xCloseGripper  := FALSE;
stMethConfig.xOpenGripper   := FALSE;

          
END_FUNCTION_BLOCK

FUNCTION_BLOCK INTERNAL FB_poweringOffState EXTENDS FB_abstractInterimMachineState

            sStateFb := __POUNAME();

stMethConfig.xGroupPowerOff := TRUE;
stMethConfig.xGroupPowerOn  := FALSE;
stMethConfig.xGroupEnable   := FALSE;
stMethConfig.xGroupDisable  := FALSE;
stMethConfig.xMoveDirAbs    := FALSE;
stMethConfig.xGroupHalt     := FALSE;
stMethConfig.xCloseGripper  := FALSE;
stMethConfig.xOpenGripper   := FALSE;

          
END_FUNCTION_BLOCK

FUNCTION_BLOCK INTERNAL FB_poweringOnState EXTENDS FB_abstractInterimMachineState

            sStateFb := __POUNAME();

stMethConfig.xGroupPowerOff := FALSE;
stMethConfig.xGroupPowerOn  := TRUE;
stMethConfig.xGroupEnable   := FALSE;
stMethConfig.xGroupDisable  := FALSE;
stMethConfig.xMoveDirAbs    := FALSE;
stMethConfig.xGroupHalt     := FALSE;
stMethConfig.xCloseGripper  := FALSE;
stMethConfig.xOpenGripper   := FALSE;

          
END_FUNCTION_BLOCK

// supposed to replicate floatToIntBits() in Java at
// https://github.com/openjdk/jdk/blob/739769c8fc4b496f08a92225a12d07414537b6c0/src/java.base/share/classes/java/lang/Float.java#L775
// , use
// https://www.exploringbinary.com/floating-point-converter/ 
// and 
// https://www.exploringbinary.com/base-converter/ 
// to double check conversion of floating point binary to base 10 integer 
// (note that website shows big endian and defaults to single precision float whereas LREAL is double precision float)
FUNCTION F_lrealToLintBits : LINT
VAR_INPUT
  lrVal : LREAL;
END_VAR
VAR
  uLrealToLintBits : U_lrealToRawLintBits; // for interpreting LREAL as base 10 LINT
END_VAR

            IF CW40.SM3_Basic.FPU.IsLRealPosInfinity(lrVal) THEN
  F_lrealToLintBits := 2139095040; // corresponds to 0x7f800000
ELSIF CW40.SM3_Basic.FPU.IsLRealNegInfinity(lrVal) THEN
  F_lrealToLintBits := 4286578688; // corresponds to 0xff800000
ELSIF CW40.SM3_Basic.FPU.IsLRealNaN(lrVal) THEN
  F_lrealToLintBits := 2143289344; // corresponds to 0x7fc00000
ELSE
  uLrealToLintBits.lrVal := lrVal;
  F_lrealToLintBits := uLrealToLintBits.liVal;
END_IF

          
END_FUNCTION

FUNCTION_BLOCK INTERNAL FB_mcMoveElement EXTENDS COL.LinkedListElementBase IMPLEMENTS I_mcMoveElement
VAR_INPUT
  stMcMoveParams : ST_mcMoveParams;
  uliMotionIndx  : ULINT;
END_VAR
VAR
  mcMoveCrcAbs : SM3_Robotics.MC_MoveCircularAbsolute;
  mcMoveCrcRel : SM3_Robotics.MC_MoveCircularRelative;
  mcMoveDirAbs : SM3_Robotics.MC_MoveDirectAbsolute;
  mcMoveDirRel : SM3_Robotics.MC_MoveDirectRelative;
  mcMoveLinAbs : SM3_Robotics.MC_MoveLinearAbsolute;
  mcMoveLinRel : SM3_Robotics.MC_MoveLinearRelative;

  fbLogAdd : FB_logAdd(pCmpName:=ADR(__POUNAME()));
END_VAR

            
          

(* Returns the hashcode of this element.
 This method is used by hash based collections (e.g. |Hashtable|) to get the hashcode from a element.
 IMPORTANT: The value of the method MUST NOT be changed during the lifecycle of the object.*)
METHOD ElementHashCode : LINT
VAR
  liPrime   : LINT := 37;
  liInitVal : LINT := 1; // has to be nonzero
END_VAR
                  // https://stackoverflow.com/questions/5443136/are-two-java-objects-with-same-hashcodes-not-necessarily-equal/5443140#5443140
// IF two objects have the same hashcode THEN they are NOT necessarily equal. Otherwise you will have discovered the perfect hash FUNCTION.
// But the opposite is true: if the objects are equal, then they must have the same hashcode.

// based on https://stackoverflow.com/questions/113511/best-implementation-for-hashcode-method-for-a-collection/113600#113600
ElementHashCode := liInitVal;

ElementHashCode := (ElementHashCode * liPrime) + ULINT_TO_LINT(uliMotionIndx);
ElementHashCode := (ElementHashCode * liPrime) + TO_LINT(stMcMoveParams.eMcMotionFbType);

CASE stMcMoveParams.eMcMotionFbType OF

  E_mcMotionFbType.moveCrcAbs:
    ElementHashCode := (ElementHashCode * liPrime) + METH_stMoveCrcParamsHashCode();
    ElementHashCode := (ElementHashCode * liPrime) + METH_mcMoveCrcAbsHashCode();

  E_mcMotionFbType.moveCrcRel:
    ElementHashCode := (ElementHashCode * liPrime) + METH_stMoveCrcParamsHashCode();
    ElementHashCode := (ElementHashCode * liPrime) + METH_mcMoveCrcRelHashCode();

  E_mcMotionFbType.moveDirAbs:
    ElementHashCode := (ElementHashCode * liPrime) + METH_stMoveDirParamsHashCode();
    ElementHashCode := (ElementHashCode * liPrime) + METH_mcMoveDirAbsHashCode();

  E_mcMotionFbType.moveDirRel:
    ElementHashCode := (ElementHashCode * liPrime) + METH_stMoveDirParamsHashCode();
    ElementHashCode := (ElementHashCode * liPrime) + METH_mcMoveDirRelHashCode();

  E_mcMotionFbType.moveLinAbs:
    ElementHashCode := (ElementHashCode * liPrime) + METH_stMoveLinParamsHashCode();
    ElementHashCode := (ElementHashCode * liPrime) + METH_mcMoveLinAbsHashCode();

  E_mcMotionFbType.moveLinRel:
    ElementHashCode := (ElementHashCode * liPrime) + METH_stMoveLinParamsHashCode();
    ElementHashCode := (ElementHashCode * liPrime) + METH_mcMoveLinRelHashCode();

END_CASE

                
END_METHOD

(* Compares this element with itfElement.
 Returns 0 if the elements are equal, < 0 if the element is less than itfElement, 
 > 0 if the element is greater than itfElement.
 This method will be called from sorted collections (e.g. |SortedList|) to sort elements.
 IMPORTANT: The underlying value to be compared with MUST NOT be changed during the lifecycle of the object.*)
METHOD ElementCompareTo : INT
VAR_INPUT
  (* The element to compare*)
  itfElement : COL.IElement;
END_VAR
VAR
  itfMcMoveElem : I_mcMoveElement; // __QUERYINTERFACE will convert to this
END_VAR
                  // default to no change when sorting
ElementCompareTo := 0;

// diMotionIndx used for sorting
IF __QUERYINTERFACE(itfElement, itfMcMoveElem) THEN
  IF (THIS^.PROP_motionIndx > itfMcMoveElem.PROP_motionIndx) THEN
    ElementCompareTo := 1;
  ELSIF (THIS^.PROP_motionIndx < itfMcMoveElem.PROP_motionIndx) THEN
    ElementCompareTo := -1;
  END_IF
END_IF

                
END_METHOD

(* Returns true of this element and itfElement are equal.
 This method will be called from the function block |HashTable| to find an element by key if the hashcode of an element collides with an other element.
 IMPORTANT: The underlying value to be compared with MUST NOT be changed during the lifecycle of the object.*)
METHOD ElementEquals : BOOL
VAR_INPUT
  (* The element to compare*)
  itfElement : COL.IElement;
END_VAR
VAR
  itfMcMoveElem : I_mcMoveElement; // __QUERYINTERFACE will convert to this

  instMcMoveParams : ST_mcMoveParams;

  lrTol : LREAL := 1E-3;
END_VAR
                  ElementEquals := FALSE;

IF __QUERYINTERFACE(itfElement, itfMcMoveElem) THEN

  IF (THIS^.uliMotionIndx <> itfMcMoveElem.PROP_motionIndx) THEN
    RETURN;
  END_IF

  instMcMoveParams := itfMcMoveElem.PROP_stMcMoveParams;

  IF (THIS^.stMcMoveParams.eMcMotionFbType <> instMcMoveParams.eMcMotionFbType) THEN
    RETURN;
  END_IF

  CASE THIS^.stMcMoveParams.eMcMotionFbType OF

    E_mcMotionFbType.moveCrcAbs:
      ElementEquals := (
        METH_stMoveCrcParamsEquals(instMcMoveParams.stMoveCrcParams, lrTol) AND METH_mcMoveCrcAbsEquals(itfMcMoveElem.PROP_mcMoveCrcAbs, lrTol)
        );

    E_mcMotionFbType.moveCrcRel:
      ElementEquals := (
        METH_stMoveCrcParamsEquals(instMcMoveParams.stMoveCrcParams, lrTol) AND METH_mcMoveCrcRelEquals(itfMcMoveElem.PROP_mcMoveCrcRel, lrTol)
        );

    E_mcMotionFbType.moveDirAbs:
      ElementEquals := (
        METH_stMoveDirParamsEquals(instMcMoveParams.stMoveDirParams, lrTol) AND METH_mcMoveDirAbsEquals(itfMcMoveElem.PROP_mcMoveDirAbs, lrTol)
        );

    E_mcMotionFbType.moveDirRel:
      ElementEquals := (
        METH_stMoveDirParamsEquals(instMcMoveParams.stMoveDirParams, lrTol) AND METH_mcMoveDirRelEquals(itfMcMoveElem.PROP_mcMoveDirRel, lrTol)
        );

    E_mcMotionFbType.moveLinAbs:
      ElementEquals := (
        METH_stMoveLinParamsEquals(instMcMoveParams.stMoveLinParams, lrTol) AND METH_mcMoveLinAbsEquals(itfMcMoveElem.PROP_mcMoveLinAbs, lrTol)
        );

    E_mcMotionFbType.moveLinRel:
      ElementEquals := (
        METH_stMoveLinParamsEquals(instMcMoveParams.stMoveLinParams, lrTol) AND METH_mcMoveLinRelEquals(itfMcMoveElem.PROP_mcMoveLinRel, lrTol)
        );

  END_CASE

END_IF

                
END_METHOD

// check only inputs of relevant MC_Move* FB
METHOD PRIVATE METH_mcMoveCrcAbsEquals : BOOL
VAR_INPUT
  inMcMoveCrcAbs : SM3_Robotics.MC_MoveCircularAbsolute;
  lrTol          : LREAL := 1E-3;
END_VAR
VAR
  diIndx : DINT;
END_VAR
                  METH_mcMoveCrcAbsEquals := FALSE;

IF (THIS^.mcMoveCrcAbs.Execute <> inMcMoveCrcAbs.Execute) THEN
  RETURN;
END_IF

IF (THIS^.mcMoveCrcAbs.CircMode <> inMcMoveCrcAbs.CircMode) THEN
  RETURN;
END_IF

FOR diIndx := LOWER_BOUND(THIS^.mcMoveCrcAbs.AuxPoint.v, 1) TO UPPER_BOUND(THIS^.mcMoveCrcAbs.AuxPoint.v, 1) BY 1 DO
  IF ABS(THIS^.mcMoveCrcAbs.AuxPoint.v[diIndx] - inMcMoveCrcAbs.AuxPoint.v[diIndx]) > lrTol THEN
    RETURN;
  END_IF
END_FOR

FOR diIndx := LOWER_BOUND(THIS^.mcMoveCrcAbs.EndPoint.v, 1) TO UPPER_BOUND(THIS^.mcMoveCrcAbs.EndPoint.v, 1) BY 1 DO
  IF ABS(THIS^.mcMoveCrcAbs.EndPoint.v[diIndx] - inMcMoveCrcAbs.EndPoint.v[diIndx]) > lrTol THEN
    RETURN;
  END_IF
END_FOR

IF (THIS^.mcMoveCrcAbs.PathChoice <> inMcMoveCrcAbs.PathChoice) THEN
  RETURN;
END_IF

IF ABS(THIS^.mcMoveCrcAbs.Velocity - inMcMoveCrcAbs.Velocity) > lrTol THEN
  RETURN;
END_IF

IF ABS(THIS^.mcMoveCrcAbs.Acceleration - inMcMoveCrcAbs.Acceleration) > lrTol THEN
  RETURN;
END_IF

IF ABS(THIS^.mcMoveCrcAbs.Deceleration - inMcMoveCrcAbs.Deceleration) > lrTol THEN
  RETURN;
END_IF

IF ABS(THIS^.mcMoveCrcAbs.Jerk - inMcMoveCrcAbs.Jerk) > lrTol THEN
  RETURN;
END_IF

IF (THIS^.mcMoveCrcAbs.CoordSystem <> inMcMoveCrcAbs.CoordSystem) THEN
  RETURN;
END_IF

IF (THIS^.mcMoveCrcAbs.BufferMode <> inMcMoveCrcAbs.BufferMode) THEN
  RETURN;
END_IF

IF (THIS^.mcMoveCrcAbs.TransitionMode <> inMcMoveCrcAbs.TransitionMode) THEN
  RETURN;
END_IF

FOR diIndx := LOWER_BOUND(THIS^.mcMoveCrcAbs.TransitionParameter, 1) TO UPPER_BOUND(THIS^.mcMoveCrcAbs.TransitionParameter, 1) DO
  IF ABS(THIS^.mcMoveCrcAbs.TransitionParameter[diIndx] - inMcMoveCrcAbs.TransitionParameter[diIndx]) > lrTol THEN
    RETURN;
  END_IF
END_FOR

IF (THIS^.mcMoveCrcAbs.OrientationMode <> inMcMoveCrcAbs.OrientationMode) THEN
  RETURN;
END_IF

IF ABS(THIS^.mcMoveCrcAbs.VelFactor - inMcMoveCrcAbs.VelFactor) > lrTol THEN
  RETURN;
END_IF

IF ABS(THIS^.mcMoveCrcAbs.AccFactor - inMcMoveCrcAbs.AccFactor) > lrTol THEN
  RETURN;
END_IF

IF ABS(THIS^.mcMoveCrcAbs.JerkFactor - inMcMoveCrcAbs.JerkFactor) > lrTol THEN
  RETURN;
END_IF

METH_mcMoveCrcAbsEquals := TRUE;

                
END_METHOD

// check only inputs of relevant MC_Move* FB
METHOD PRIVATE METH_mcMoveDirAbsEquals : BOOL
VAR_INPUT
  inMcMoveDirAbs : SM3_Robotics.MC_MoveDirectAbsolute;
  lrTol          : LREAL := 1E-3;
END_VAR
VAR
  diIndx : DINT;
END_VAR
                  METH_mcMoveDirAbsEquals := FALSE;

IF (THIS^.mcMoveDirAbs.Execute <> inMcMoveDirAbs.Execute) THEN
  RETURN;
END_IF

FOR diIndx := LOWER_BOUND(THIS^.mcMoveDirAbs.Position.v, 1) TO UPPER_BOUND(THIS^.mcMoveDirAbs.Position.v, 1) BY 1 DO
  IF ABS(THIS^.mcMoveDirAbs.Position.v[diIndx] - inMcMoveDirAbs.Position.v[diIndx]) > lrTol THEN
    RETURN;
  END_IF
END_FOR

IF (THIS^.mcMoveDirAbs.MovementType <> inMcMoveDirAbs.MovementType) THEN
  RETURN;
END_IF

IF (THIS^.mcMoveDirAbs.CoordSystem <> inMcMoveDirAbs.CoordSystem) THEN
  RETURN;
END_IF

IF (THIS^.mcMoveDirAbs.BufferMode <> inMcMoveDirAbs.BufferMode) THEN
  RETURN;
END_IF

IF (THIS^.mcMoveDirAbs.TransitionMode <> inMcMoveDirAbs.TransitionMode) THEN
  RETURN;
END_IF

FOR diIndx := LOWER_BOUND(THIS^.mcMoveDirAbs.TransitionParameter, 1) TO UPPER_BOUND(THIS^.mcMoveDirAbs.TransitionParameter, 1) DO
  IF ABS(THIS^.mcMoveDirAbs.TransitionParameter[diIndx] - inMcMoveDirAbs.TransitionParameter[diIndx]) > lrTol THEN
    RETURN;
  END_IF
END_FOR

IF ABS(THIS^.mcMoveDirAbs.VelFactor - inMcMoveDirAbs.VelFactor) > lrTol THEN
  RETURN;
END_IF

IF ABS(THIS^.mcMoveDirAbs.AccFactor - inMcMoveDirAbs.AccFactor) > lrTol THEN
  RETURN;
END_IF

IF ABS(THIS^.mcMoveDirAbs.JerkFactor - inMcMoveDirAbs.JerkFactor) > lrTol THEN
  RETURN;
END_IF

METH_mcMoveDirAbsEquals := TRUE;

                
END_METHOD

// based on https://stackoverflow.com/questions/113511/best-implementation-for-hashcode-method-for-a-collection/113600#113600
METHOD PRIVATE METH_stMoveDirParamsHashCode : LINT
VAR_INPUT
  liPrime : LINT := 37;
END_VAR
VAR
  liInitVal : LINT := 1; // has to be nonzero
  diIndx    : DINT;
END_VAR
                  METH_stMoveDirParamsHashCode := liInitVal;

FOR diIndx := LOWER_BOUND(stMcMoveParams.stMoveDirParams.smcPosRef.v, 1) TO
  UPPER_BOUND(stMcMoveParams.stMoveDirParams.smcPosRef.v, 1) BY 1 DO
  METH_stMoveDirParamsHashCode :=
    (METH_stMoveDirParamsHashCode * liPrime) + F_lrealToLintBits(stMcMoveParams.stMoveDirParams.smcPosRef.v[diIndx]);
END_FOR

METH_stMoveDirParamsHashCode := (METH_stMoveDirParamsHashCode * liPrime) + TO_LINT(stMcMoveParams.stMoveDirParams.smcPtpTyp);

METH_stMoveDirParamsHashCode := (METH_stMoveDirParamsHashCode * liPrime) + TO_LINT(stMcMoveParams.stMoveDirParams.smcCrdSys);

METH_stMoveDirParamsHashCode := (METH_stMoveDirParamsHashCode * liPrime) + TO_LINT(stMcMoveParams.stMoveDirParams.mcBufMode);

METH_stMoveDirParamsHashCode := (METH_stMoveDirParamsHashCode * liPrime) + TO_LINT(stMcMoveParams.stMoveDirParams.mcTrnMode);

FOR diIndx := LOWER_BOUND(stMcMoveParams.stMoveDirParams.arrTrnPrm, 1) TO
  UPPER_BOUND(stMcMoveParams.stMoveDirParams.arrTrnPrm, 1) BY 1 DO
  METH_stMoveDirParamsHashCode :=
    (METH_stMoveDirParamsHashCode * liPrime) + F_lrealToLintBits(stMcMoveParams.stMoveDirParams.arrTrnPrm[diIndx]);
END_FOR

METH_stMoveDirParamsHashCode := (METH_stMoveDirParamsHashCode * liPrime) + F_lrealToLintBits(stMcMoveParams.stMoveDirParams.lrVelFctr);

METH_stMoveDirParamsHashCode := (METH_stMoveDirParamsHashCode * liPrime) + F_lrealToLintBits(stMcMoveParams.stMoveDirParams.lrAccFctr);

METH_stMoveDirParamsHashCode := (METH_stMoveDirParamsHashCode * liPrime) + F_lrealToLintBits(stMcMoveParams.stMoveDirParams.lrJrkFctr);

                
END_METHOD

// check only inputs of relevant MC_Move* FB
METHOD PRIVATE METH_mcMoveDirRelEquals : BOOL
VAR_INPUT
  inMcMoveDirRel : SM3_Robotics.MC_MoveDirectRelative;
  lrTol          : LREAL := 1E-3;
END_VAR
VAR
  diIndx : DINT;
END_VAR
                  METH_mcMoveDirRelEquals := FALSE;

IF (THIS^.mcMoveDirRel.Execute <> inMcMoveDirRel.Execute) THEN
  RETURN;
END_IF

FOR diIndx := LOWER_BOUND(THIS^.mcMoveDirRel.Distance.v, 1) TO UPPER_BOUND(THIS^.mcMoveDirRel.Distance.v, 1) BY 1 DO
  IF ABS(THIS^.mcMoveDirRel.Distance.v[diIndx] - inMcMoveDirRel.Distance.v[diIndx]) > lrTol THEN
    RETURN;
  END_IF
END_FOR

IF (THIS^.mcMoveDirRel.MovementType <> inMcMoveDirRel.MovementType) THEN
  RETURN;
END_IF

IF (THIS^.mcMoveDirRel.CoordSystem <> inMcMoveDirRel.CoordSystem) THEN
  RETURN;
END_IF

IF (THIS^.mcMoveDirRel.BufferMode <> inMcMoveDirRel.BufferMode) THEN
  RETURN;
END_IF

IF (THIS^.mcMoveDirRel.TransitionMode <> inMcMoveDirRel.TransitionMode) THEN
  RETURN;
END_IF

FOR diIndx := LOWER_BOUND(THIS^.mcMoveDirRel.TransitionParameter, 1) TO UPPER_BOUND(THIS^.mcMoveDirRel.TransitionParameter, 1) DO
  IF ABS(THIS^.mcMoveDirRel.TransitionParameter[diIndx] - inMcMoveDirRel.TransitionParameter[diIndx]) > lrTol THEN
    RETURN;
  END_IF
END_FOR

IF ABS(THIS^.mcMoveDirRel.VelFactor - inMcMoveDirRel.VelFactor) > lrTol THEN
  RETURN;
END_IF

IF ABS(THIS^.mcMoveDirRel.AccFactor - inMcMoveDirRel.AccFactor) > lrTol THEN
  RETURN;
END_IF

IF ABS(THIS^.mcMoveDirRel.JerkFactor - inMcMoveDirRel.JerkFactor) > lrTol THEN
  RETURN;
END_IF

METH_mcMoveDirRelEquals := TRUE;

                
END_METHOD

// check only inputs of relevant MC_Move* FB
METHOD PRIVATE METH_mcMoveCrcRelEquals : BOOL
VAR_INPUT
  inMcMoveCrcRel : SM3_Robotics.MC_MoveCircularRelative;
  lrTol          : LREAL := 1E-3;
END_VAR
VAR
  diIndx : DINT;
END_VAR
                  METH_mcMoveCrcRelEquals := FALSE;

IF (THIS^.mcMoveCrcRel.Execute <> inMcMoveCrcRel.Execute) THEN
  RETURN;
END_IF

IF (THIS^.mcMoveCrcRel.CircMode <> inMcMoveCrcRel.CircMode) THEN
  RETURN;
END_IF

FOR diIndx := LOWER_BOUND(THIS^.mcMoveCrcRel.AuxPoint.v, 1) TO UPPER_BOUND(THIS^.mcMoveCrcRel.AuxPoint.v, 1) BY 1 DO
  IF ABS(THIS^.mcMoveCrcRel.AuxPoint.v[diIndx] - inMcMoveCrcRel.AuxPoint.v[diIndx]) > lrTol THEN
    RETURN;
  END_IF
END_FOR

FOR diIndx := LOWER_BOUND(THIS^.mcMoveCrcRel.EndPoint.v, 1) TO UPPER_BOUND(THIS^.mcMoveCrcRel.EndPoint.v, 1) BY 1 DO
  IF ABS(THIS^.mcMoveCrcRel.EndPoint.v[diIndx] - inMcMoveCrcRel.EndPoint.v[diIndx]) > lrTol THEN
    RETURN;
  END_IF
END_FOR

IF (THIS^.mcMoveCrcRel.PathChoice <> inMcMoveCrcRel.PathChoice) THEN
  RETURN;
END_IF

IF ABS(THIS^.mcMoveCrcRel.Velocity - inMcMoveCrcRel.Velocity) > lrTol THEN
  RETURN;
END_IF

IF ABS(THIS^.mcMoveCrcRel.Acceleration - inMcMoveCrcRel.Acceleration) > lrTol THEN
  RETURN;
END_IF

IF ABS(THIS^.mcMoveCrcRel.Deceleration - inMcMoveCrcRel.Deceleration) > lrTol THEN
  RETURN;
END_IF

IF ABS(THIS^.mcMoveCrcRel.Jerk - inMcMoveCrcRel.Jerk) > lrTol THEN
  RETURN;
END_IF

IF (THIS^.mcMoveCrcRel.CoordSystem <> inMcMoveCrcRel.CoordSystem) THEN
  RETURN;
END_IF

IF (THIS^.mcMoveCrcRel.BufferMode <> inMcMoveCrcRel.BufferMode) THEN
  RETURN;
END_IF

IF (THIS^.mcMoveCrcRel.TransitionMode <> inMcMoveCrcRel.TransitionMode) THEN
  RETURN;
END_IF

FOR diIndx := LOWER_BOUND(THIS^.mcMoveCrcRel.TransitionParameter, 1) TO UPPER_BOUND(THIS^.mcMoveCrcRel.TransitionParameter, 1) DO
  IF ABS(THIS^.mcMoveCrcRel.TransitionParameter[diIndx] - inMcMoveCrcRel.TransitionParameter[diIndx]) > lrTol THEN
    RETURN;
  END_IF
END_FOR

IF (THIS^.mcMoveCrcRel.OrientationMode <> inMcMoveCrcRel.OrientationMode) THEN
  RETURN;
END_IF

IF ABS(THIS^.mcMoveCrcRel.VelFactor - inMcMoveCrcRel.VelFactor) > lrTol THEN
  RETURN;
END_IF

IF ABS(THIS^.mcMoveCrcRel.AccFactor - inMcMoveCrcRel.AccFactor) > lrTol THEN
  RETURN;
END_IF

IF ABS(THIS^.mcMoveCrcRel.JerkFactor - inMcMoveCrcRel.JerkFactor) > lrTol THEN
  RETURN;
END_IF

METH_mcMoveCrcRelEquals := TRUE;

                
END_METHOD

// check only inputs of relevant MC_Move* FB
METHOD PRIVATE METH_mcMoveLinAbsEquals : BOOL
VAR_INPUT
  inMcMoveLinAbs : SM3_Robotics.MC_MoveLinearAbsolute;
  lrTol          : LREAL := 1E-3;
END_VAR
VAR
  diIndx : DINT;
END_VAR
                  METH_mcMoveLinAbsEquals := FALSE;

IF (THIS^.mcMoveLinAbs.Execute <> inMcMoveLinAbs.Execute) THEN
  RETURN;
END_IF

FOR diIndx := LOWER_BOUND(THIS^.mcMoveLinAbs.Position.v, 1) TO UPPER_BOUND(THIS^.mcMoveLinAbs.Position.v, 1) BY 1 DO
  IF ABS(THIS^.mcMoveLinAbs.Position.v[diIndx] - inMcMoveLinAbs.Position.v[diIndx]) > lrTol THEN
    RETURN;
  END_IF
END_FOR

IF ABS(THIS^.mcMoveLinAbs.Velocity - inMcMoveLinAbs.Velocity) > lrTol THEN
  RETURN;
END_IF

IF ABS(THIS^.mcMoveLinAbs.Acceleration - inMcMoveLinAbs.Acceleration) > lrTol THEN
  RETURN;
END_IF

IF ABS(THIS^.mcMoveLinAbs.Deceleration - inMcMoveLinAbs.Deceleration) > lrTol THEN
  RETURN;
END_IF

IF ABS(THIS^.mcMoveLinAbs.Jerk - inMcMoveLinAbs.Jerk) > lrTol THEN
  RETURN;
END_IF

IF (THIS^.mcMoveLinAbs.CoordSystem <> inMcMoveLinAbs.CoordSystem) THEN
  RETURN;
END_IF

IF (THIS^.mcMoveLinAbs.BufferMode <> inMcMoveLinAbs.BufferMode) THEN
  RETURN;
END_IF

IF (THIS^.mcMoveLinAbs.TransitionMode <> inMcMoveLinAbs.TransitionMode) THEN
  RETURN;
END_IF

FOR diIndx := LOWER_BOUND(THIS^.mcMoveLinAbs.TransitionParameter, 1) TO UPPER_BOUND(THIS^.mcMoveLinAbs.TransitionParameter, 1) DO
  IF ABS(THIS^.mcMoveLinAbs.TransitionParameter[diIndx] - inMcMoveLinAbs.TransitionParameter[diIndx]) > lrTol THEN
    RETURN;
  END_IF
END_FOR

IF (THIS^.mcMoveLinAbs.OrientationMode <> inMcMoveLinAbs.OrientationMode) THEN
  RETURN;
END_IF

IF ABS(THIS^.mcMoveLinAbs.VelFactor - inMcMoveLinAbs.VelFactor) > lrTol THEN
  RETURN;
END_IF

IF ABS(THIS^.mcMoveLinAbs.AccFactor - inMcMoveLinAbs.AccFactor) > lrTol THEN
  RETURN;
END_IF

IF ABS(THIS^.mcMoveLinAbs.JerkFactor - inMcMoveLinAbs.JerkFactor) > lrTol THEN
  RETURN;
END_IF

METH_mcMoveLinAbsEquals := TRUE;

                
END_METHOD

// check only inputs of relevant MC_Move* FB
METHOD PRIVATE METH_mcMoveLinRelEquals : BOOL
VAR_INPUT
  inMcMoveLinRel : SM3_Robotics.MC_MoveLinearRelative;
  lrTol          : LREAL := 1E-3;
END_VAR
VAR
  diIndx : DINT;
END_VAR
                  METH_mcMoveLinRelEquals := FALSE;

IF (THIS^.mcMoveLinRel.Execute <> inMcMoveLinRel.Execute) THEN
  RETURN;
END_IF

FOR diIndx := LOWER_BOUND(THIS^.mcMoveLinRel.Distance.v, 1) TO UPPER_BOUND(THIS^.mcMoveLinRel.Distance.v, 1) BY 1 DO
  IF ABS(THIS^.mcMoveLinRel.Distance.v[diIndx] - inMcMoveLinRel.Distance.v[diIndx]) > lrTol THEN
    RETURN;
  END_IF
END_FOR

IF ABS(THIS^.mcMoveLinRel.Velocity - inMcMoveLinRel.Velocity) > lrTol THEN
  RETURN;
END_IF

IF ABS(THIS^.mcMoveLinRel.Acceleration - inMcMoveLinRel.Acceleration) > lrTol THEN
  RETURN;
END_IF

IF ABS(THIS^.mcMoveLinRel.Deceleration - inMcMoveLinRel.Deceleration) > lrTol THEN
  RETURN;
END_IF

IF ABS(THIS^.mcMoveLinRel.Jerk - inMcMoveLinRel.Jerk) > lrTol THEN
  RETURN;
END_IF

IF (THIS^.mcMoveLinRel.CoordSystem <> inMcMoveLinRel.CoordSystem) THEN
  RETURN;
END_IF

IF (THIS^.mcMoveLinRel.BufferMode <> inMcMoveLinRel.BufferMode) THEN
  RETURN;
END_IF

IF (THIS^.mcMoveLinRel.TransitionMode <> inMcMoveLinRel.TransitionMode) THEN
  RETURN;
END_IF

FOR diIndx := LOWER_BOUND(THIS^.mcMoveLinRel.TransitionParameter, 1) TO UPPER_BOUND(THIS^.mcMoveLinRel.TransitionParameter, 1) DO
  IF ABS(THIS^.mcMoveLinRel.TransitionParameter[diIndx] - inMcMoveLinRel.TransitionParameter[diIndx]) > lrTol THEN
    RETURN;
  END_IF
END_FOR

IF (THIS^.mcMoveLinRel.OrientationMode <> inMcMoveLinRel.OrientationMode) THEN
  RETURN;
END_IF

IF ABS(THIS^.mcMoveLinRel.VelFactor - inMcMoveLinRel.VelFactor) > lrTol THEN
  RETURN;
END_IF

IF ABS(THIS^.mcMoveLinRel.AccFactor - inMcMoveLinRel.AccFactor) > lrTol THEN
  RETURN;
END_IF

IF ABS(THIS^.mcMoveLinRel.JerkFactor - inMcMoveLinRel.JerkFactor) > lrTol THEN
  RETURN;
END_IF

METH_mcMoveLinRelEquals := TRUE;

                
END_METHOD

// based on https://stackoverflow.com/questions/113511/best-implementation-for-hashcode-method-for-a-collection/113600#113600
METHOD PRIVATE METH_mcMoveCrcAbsHashCode : LINT
VAR_INPUT
  liPrime : LINT := 37;
END_VAR
VAR
  liInitVal : LINT := 1; // has to be nonzero
  diIndx    : DINT;
END_VAR
                  METH_mcMoveCrcAbsHashCode := liInitVal;

METH_mcMoveCrcAbsHashCode := (METH_mcMoveCrcAbsHashCode * liPrime) + BOOL_TO_LINT(mcMoveCrcAbs.Execute);

METH_mcMoveCrcAbsHashCode := (METH_mcMoveCrcAbsHashCode * liPrime) + TO_LINT(mcMoveCrcAbs.CircMode);

FOR diIndx := LOWER_BOUND(mcMoveCrcAbs.AuxPoint.v, 1) TO UPPER_BOUND(mcMoveCrcAbs.AuxPoint.v, 1) BY 1 DO
  METH_mcMoveCrcAbsHashCode := (METH_mcMoveCrcAbsHashCode * liPrime) + F_lrealToLintBits(mcMoveCrcAbs.AuxPoint.v[diIndx]);
END_FOR

FOR diIndx := LOWER_BOUND(mcMoveCrcAbs.EndPoint.v, 1) TO UPPER_BOUND(mcMoveCrcAbs.EndPoint.v, 1) BY 1 DO
  METH_mcMoveCrcAbsHashCode := (METH_mcMoveCrcAbsHashCode * liPrime) + F_lrealToLintBits(mcMoveCrcAbs.EndPoint.v[diIndx]);
END_FOR

METH_mcMoveCrcAbsHashCode := (METH_mcMoveCrcAbsHashCode * liPrime) + TO_LINT(mcMoveCrcAbs.PathChoice);

METH_mcMoveCrcAbsHashCode := (METH_mcMoveCrcAbsHashCode * liPrime) + F_lrealToLintBits(mcMoveCrcAbs.Velocity);

METH_mcMoveCrcAbsHashCode := (METH_mcMoveCrcAbsHashCode * liPrime) + F_lrealToLintBits(mcMoveCrcAbs.Acceleration);

METH_mcMoveCrcAbsHashCode := (METH_mcMoveCrcAbsHashCode * liPrime) + F_lrealToLintBits(mcMoveCrcAbs.Deceleration);

METH_mcMoveCrcAbsHashCode := (METH_mcMoveCrcAbsHashCode * liPrime) + F_lrealToLintBits(mcMoveCrcAbs.Jerk);

METH_mcMoveCrcAbsHashCode := (METH_mcMoveCrcAbsHashCode * liPrime) + TO_LINT(mcMoveCrcAbs.CoordSystem);

METH_mcMoveCrcAbsHashCode := (METH_mcMoveCrcAbsHashCode * liPrime) + TO_LINT(mcMoveCrcAbs.BufferMode);

METH_mcMoveCrcAbsHashCode := (METH_mcMoveCrcAbsHashCode * liPrime) + TO_LINT(mcMoveCrcAbs.TransitionMode);

FOR diIndx := LOWER_BOUND(mcMoveCrcAbs.TransitionParameter, 1) TO UPPER_BOUND(mcMoveCrcAbs.TransitionParameter, 1) BY 1 DO
  METH_mcMoveCrcAbsHashCode := (METH_mcMoveCrcAbsHashCode * liPrime) + F_lrealToLintBits(mcMoveCrcAbs.TransitionParameter[diIndx]);
END_FOR

METH_mcMoveCrcAbsHashCode := (METH_mcMoveCrcAbsHashCode * liPrime) + TO_LINT(mcMoveCrcAbs.OrientationMode);

METH_mcMoveCrcAbsHashCode := (METH_mcMoveCrcAbsHashCode * liPrime) + F_lrealToLintBits(mcMoveCrcAbs.VelFactor);

METH_mcMoveCrcAbsHashCode := (METH_mcMoveCrcAbsHashCode * liPrime) + F_lrealToLintBits(mcMoveCrcAbs.AccFactor);

METH_mcMoveCrcAbsHashCode := (METH_mcMoveCrcAbsHashCode * liPrime) + F_lrealToLintBits(mcMoveCrcAbs.JerkFactor);

                
END_METHOD

// check motion parameters in relevant struct
METHOD PRIVATE METH_stMoveCrcParamsEquals : BOOL
VAR_INPUT
  inStMoveCrcParams : ST_moveCrcParams;
  lrTol             : LREAL := 1E-3;
END_VAR
VAR
  diIndx : DINT;
END_VAR
                  METH_stMoveCrcParamsEquals := FALSE;

IF (THIS^.stMcMoveParams.stMoveCrcParams.smcCrcMod <> inStMoveCrcParams.smcCrcMod) THEN
  RETURN;
END_IF

FOR diIndx := LOWER_BOUND(THIS^.stMcMoveParams.stMoveCrcParams.smcPosRef_auxPt.v, 1) TO
  UPPER_BOUND(THIS^.stMcMoveParams.stMoveCrcParams.smcPosRef_auxPt.v, 1) BY 1 DO
  IF ABS(THIS^.stMcMoveParams.stMoveCrcParams.smcPosRef_auxPt.v[diIndx] - inStMoveCrcParams.smcPosRef_auxPt.v[diIndx]) > lrTol THEN
    RETURN;
  END_IF
END_FOR

FOR diIndx := LOWER_BOUND(THIS^.stMcMoveParams.stMoveCrcParams.smcPosRef_endPt.v, 1) TO
  UPPER_BOUND(THIS^.stMcMoveParams.stMoveCrcParams.smcPosRef_endPt.v, 1) BY 1 DO
  IF ABS(THIS^.stMcMoveParams.stMoveCrcParams.smcPosRef_endPt.v[diIndx] - inStMoveCrcParams.smcPosRef_endPt.v[diIndx]) > lrTol THEN
    RETURN;
  END_IF
END_FOR

IF (THIS^.stMcMoveParams.stMoveCrcParams.mcCrcPathChoice <> inStMoveCrcParams.mcCrcPathChoice) THEN
  RETURN;
END_IF

IF ABS(THIS^.stMcMoveParams.stMoveCrcParams.lrVel - inStMoveCrcParams.lrVel) > lrTol THEN
  RETURN;
END_IF

IF ABS(THIS^.stMcMoveParams.stMoveCrcParams.lrAcc - inStMoveCrcParams.lrAcc) > lrTol THEN
  RETURN;
END_IF

IF ABS(THIS^.stMcMoveParams.stMoveCrcParams.lrDec - inStMoveCrcParams.lrDec) > lrTol THEN
  RETURN;
END_IF

IF ABS(THIS^.stMcMoveParams.stMoveCrcParams.lrJrk - inStMoveCrcParams.lrJrk) > lrTol THEN
  RETURN;
END_IF

IF (THIS^.stMcMoveParams.stMoveCrcParams.smcCrdSys <> inStMoveCrcParams.smcCrdSys) THEN
  RETURN;
END_IF

IF (THIS^.stMcMoveParams.stMoveCrcParams.mcBufMode <> inStMoveCrcParams.mcBufMode) THEN
  RETURN;
END_IF

IF (THIS^.stMcMoveParams.stMoveCrcParams.mcTrnMode <> inStMoveCrcParams.mcTrnMode) THEN
  RETURN;
END_IF

FOR diIndx :=
  LOWER_BOUND(THIS^.stMcMoveParams.stMoveCrcParams.arrTrnPrm, 1) TO UPPER_BOUND(THIS^.stMcMoveParams.stMoveCrcParams.arrTrnPrm, 1) BY 1 DO
  IF ABS(THIS^.stMcMoveParams.stMoveCrcParams.arrTrnPrm[diIndx] - inStMoveCrcParams.arrTrnPrm[diIndx]) > lrTol THEN
    RETURN;
  END_IF
END_FOR

IF (THIS^.stMcMoveParams.stMoveCrcParams.smcOrnMod <> inStMoveCrcParams.smcOrnMod) THEN
  RETURN;
END_IF

IF ABS(THIS^.stMcMoveParams.stMoveCrcParams.lrVelFctr - inStMoveCrcParams.lrVelFctr) > lrTol THEN
  RETURN;
END_IF

IF ABS(THIS^.stMcMoveParams.stMoveCrcParams.lrAccFctr - inStMoveCrcParams.lrAccFctr) > lrTol THEN
  RETURN;
END_IF

IF ABS(THIS^.stMcMoveParams.stMoveCrcParams.lrJrkFctr - inStMoveCrcParams.lrJrkFctr) > lrTol THEN
  RETURN;
END_IF

METH_stMoveCrcParamsEquals := TRUE;

                
END_METHOD

// check motion parameters in relevant struct
METHOD PRIVATE METH_stMoveDirParamsEquals : BOOL
VAR_INPUT
  inStMoveDirParams : ST_moveDirParams;
  lrTol             : LREAL := 1E-3;
END_VAR
VAR
  diIndx : DINT;
END_VAR
                  METH_stMoveDirParamsEquals := FALSE;

FOR diIndx := LOWER_BOUND(THIS^.stMcMoveParams.stMoveDirParams.smcPosRef.v, 1) TO
  UPPER_BOUND(THIS^.stMcMoveParams.stMoveDirParams.smcPosRef.v, 1) BY 1 DO
  IF ABS(THIS^.stMcMoveParams.stMoveDirParams.smcPosRef.v[diIndx] - inStMoveDirParams.smcPosRef.v[diIndx]) > lrTol THEN
    RETURN;
  END_IF
END_FOR

IF (THIS^.stMcMoveParams.stMoveDirParams.smcPtpTyp <> inStMoveDirParams.smcPtpTyp) THEN
  RETURN;
END_IF

IF (THIS^.stMcMoveParams.stMoveDirParams.smcCrdSys <> inStMoveDirParams.smcCrdSys) THEN
  RETURN;
END_IF

IF (THIS^.stMcMoveParams.stMoveDirParams.mcBufMode <> inStMoveDirParams.mcBufMode) THEN
  RETURN;
END_IF

IF (THIS^.stMcMoveParams.stMoveDirParams.mcTrnMode <> inStMoveDirParams.mcTrnMode) THEN
  RETURN;
END_IF

FOR diIndx :=
  LOWER_BOUND(THIS^.stMcMoveParams.stMoveDirParams.arrTrnPrm, 1) TO UPPER_BOUND(THIS^.stMcMoveParams.stMoveDirParams.arrTrnPrm, 1) BY 1 DO
  IF ABS(THIS^.stMcMoveParams.stMoveDirParams.arrTrnPrm[diIndx] - inStMoveDirParams.arrTrnPrm[diIndx]) > lrTol THEN
    RETURN;
  END_IF
END_FOR

IF ABS(THIS^.stMcMoveParams.stMoveDirParams.lrVelFctr - inStMoveDirParams.lrVelFctr) > lrTol THEN
  RETURN;
END_IF

IF ABS(THIS^.stMcMoveParams.stMoveDirParams.lrAccFctr - inStMoveDirParams.lrAccFctr) > lrTol THEN
  RETURN;
END_IF

IF ABS(THIS^.stMcMoveParams.stMoveDirParams.lrJrkFctr - inStMoveDirParams.lrJrkFctr) > lrTol THEN
  RETURN;
END_IF

METH_stMoveDirParamsEquals := TRUE;

                
END_METHOD

// check motion parameters in relevant struct
METHOD PRIVATE METH_stMoveLinParamsEquals : BOOL
VAR_INPUT
  inStMoveLinParams : ST_moveLinParams;
  lrTol             : LREAL := 1E-3;
END_VAR
VAR
  diIndx : DINT;
END_VAR
                  METH_stMoveLinParamsEquals := FALSE;

FOR diIndx := LOWER_BOUND(THIS^.stMcMoveParams.stMoveLinParams.smcPosRef.v, 1) TO
  UPPER_BOUND(THIS^.stMcMoveParams.stMoveLinParams.smcPosRef.v, 1) BY 1 DO
  IF ABS(THIS^.stMcMoveParams.stMoveLinParams.smcPosRef.v[diIndx] - inStMoveLinParams.smcPosRef.v[diIndx]) > lrTol THEN
    RETURN;
  END_IF
END_FOR

IF ABS(THIS^.stMcMoveParams.stMoveLinParams.lrVel - inStMoveLinParams.lrVel) > lrTol THEN
  RETURN;
END_IF

IF ABS(THIS^.stMcMoveParams.stMoveLinParams.lrAcc - inStMoveLinParams.lrAcc) > lrTol THEN
  RETURN;
END_IF

IF ABS(THIS^.stMcMoveParams.stMoveLinParams.lrDec - inStMoveLinParams.lrDec) > lrTol THEN
  RETURN;
END_IF

IF ABS(THIS^.stMcMoveParams.stMoveLinParams.lrJrk - inStMoveLinParams.lrJrk) > lrTol THEN
  RETURN;
END_IF

IF (THIS^.stMcMoveParams.stMoveLinParams.smcCrdSys <> inStMoveLinParams.smcCrdSys) THEN
  RETURN;
END_IF

IF (THIS^.stMcMoveParams.stMoveLinParams.mcBufMode <> inStMoveLinParams.mcBufMode) THEN
  RETURN;
END_IF

IF (THIS^.stMcMoveParams.stMoveLinParams.mcTrnMode <> inStMoveLinParams.mcTrnMode) THEN
  RETURN;
END_IF

FOR diIndx :=
  LOWER_BOUND(THIS^.stMcMoveParams.stMoveLinParams.arrTrnPrm, 1) TO UPPER_BOUND(THIS^.stMcMoveParams.stMoveLinParams.arrTrnPrm, 1) BY 1 DO
  IF ABS(THIS^.stMcMoveParams.stMoveLinParams.arrTrnPrm[diIndx] - inStMoveLinParams.arrTrnPrm[diIndx]) > lrTol THEN
    RETURN;
  END_IF
END_FOR

IF ABS(THIS^.stMcMoveParams.stMoveLinParams.lrVelFctr - inStMoveLinParams.lrVelFctr) > lrTol THEN
  RETURN;
END_IF

IF ABS(THIS^.stMcMoveParams.stMoveLinParams.lrAccFctr - inStMoveLinParams.lrAccFctr) > lrTol THEN
  RETURN;
END_IF

IF ABS(THIS^.stMcMoveParams.stMoveLinParams.lrJrkFctr - inStMoveLinParams.lrJrkFctr) > lrTol THEN
  RETURN;
END_IF

METH_stMoveLinParamsEquals := TRUE;

                
END_METHOD

// based on https://stackoverflow.com/questions/113511/best-implementation-for-hashcode-method-for-a-collection/113600#113600
METHOD PRIVATE METH_stMoveCrcParamsHashCode : LINT
VAR_INPUT
  liPrime : LINT := 37;
END_VAR
VAR
  liInitVal : LINT := 1; // has to be nonzero
  diIndx    : DINT;
END_VAR
                  METH_stMoveCrcParamsHashCode := liInitVal;

METH_stMoveCrcParamsHashCode := (METH_stMoveCrcParamsHashCode * liPrime) + TO_LINT(stMcMoveParams.stMoveCrcParams.smcCrcMod);

FOR diIndx := LOWER_BOUND(stMcMoveParams.stMoveCrcParams.smcPosRef_auxPt.v, 1) TO
  UPPER_BOUND(stMcMoveParams.stMoveCrcParams.smcPosRef_auxPt.v, 1) BY 1 DO
  METH_stMoveCrcParamsHashCode :=
    (METH_stMoveCrcParamsHashCode * liPrime) + F_lrealToLintBits(stMcMoveParams.stMoveCrcParams.smcPosRef_auxPt.v[diIndx]);
END_FOR

FOR diIndx := LOWER_BOUND(stMcMoveParams.stMoveCrcParams.smcPosRef_endPt.v, 1) TO
  UPPER_BOUND(stMcMoveParams.stMoveCrcParams.smcPosRef_endPt.v, 1) BY 1 DO
  METH_stMoveCrcParamsHashCode :=
    (METH_stMoveCrcParamsHashCode * liPrime) + F_lrealToLintBits(stMcMoveParams.stMoveCrcParams.smcPosRef_endPt.v[diIndx]);
END_FOR

METH_stMoveCrcParamsHashCode := (METH_stMoveCrcParamsHashCode * liPrime) + TO_LINT(stMcMoveParams.stMoveCrcParams.mcCrcPathChoice);

METH_stMoveCrcParamsHashCode := (METH_stMoveCrcParamsHashCode * liPrime) + F_lrealToLintBits(stMcMoveParams.stMoveCrcParams.lrVel);

METH_stMoveCrcParamsHashCode := (METH_stMoveCrcParamsHashCode * liPrime) + F_lrealToLintBits(stMcMoveParams.stMoveCrcParams.lrAcc);

METH_stMoveCrcParamsHashCode := (METH_stMoveCrcParamsHashCode * liPrime) + F_lrealToLintBits(stMcMoveParams.stMoveCrcParams.lrDec);

METH_stMoveCrcParamsHashCode := (METH_stMoveCrcParamsHashCode * liPrime) + F_lrealToLintBits(stMcMoveParams.stMoveCrcParams.lrJrk);

METH_stMoveCrcParamsHashCode := (METH_stMoveCrcParamsHashCode * liPrime) + TO_LINT(stMcMoveParams.stMoveCrcParams.smcCrdSys);

METH_stMoveCrcParamsHashCode := (METH_stMoveCrcParamsHashCode * liPrime) + TO_LINT(stMcMoveParams.stMoveCrcParams.mcBufMode);

METH_stMoveCrcParamsHashCode := (METH_stMoveCrcParamsHashCode * liPrime) + TO_LINT(stMcMoveParams.stMoveCrcParams.mcTrnMode);

FOR diIndx := LOWER_BOUND(stMcMoveParams.stMoveCrcParams.arrTrnPrm, 1) TO UPPER_BOUND(stMcMoveParams.stMoveCrcParams.arrTrnPrm, 1) BY 1 DO
  METH_stMoveCrcParamsHashCode := (METH_stMoveCrcParamsHashCode * liPrime) + F_lrealToLintBits(stMcMoveParams.stMoveCrcParams.arrTrnPrm[diIndx]);
END_FOR

METH_stMoveCrcParamsHashCode := (METH_stMoveCrcParamsHashCode * liPrime) + TO_LINT(stMcMoveParams.stMoveCrcParams.smcOrnMod);

METH_stMoveCrcParamsHashCode := (METH_stMoveCrcParamsHashCode * liPrime) + F_lrealToLintBits(stMcMoveParams.stMoveCrcParams.lrVelFctr);

METH_stMoveCrcParamsHashCode := (METH_stMoveCrcParamsHashCode * liPrime) + F_lrealToLintBits(stMcMoveParams.stMoveCrcParams.lrAccFctr);

METH_stMoveCrcParamsHashCode := (METH_stMoveCrcParamsHashCode * liPrime) + F_lrealToLintBits(stMcMoveParams.stMoveCrcParams.lrJrkFctr);

                
END_METHOD

// based on https://stackoverflow.com/questions/113511/best-implementation-for-hashcode-method-for-a-collection/113600#113600
METHOD PRIVATE METH_stMoveLinParamsHashCode : LINT
VAR_INPUT
  liPrime : LINT := 37;
END_VAR
VAR
  liInitVal : LINT := 1; // has to be nonzero
  diIndx    : DINT;
END_VAR
                  METH_stMoveLinParamsHashCode := liInitVal;

FOR diIndx := LOWER_BOUND(stMcMoveParams.stMoveLinParams.smcPosRef.v, 1) TO
  UPPER_BOUND(stMcMoveParams.stMoveLinParams.smcPosRef.v, 1) BY 1 DO
  METH_stMoveLinParamsHashCode :=
    (METH_stMoveLinParamsHashCode * liPrime) + F_lrealToLintBits(stMcMoveParams.stMoveLinParams.smcPosRef.v[diIndx]);
END_FOR

METH_stMoveLinParamsHashCode := (METH_stMoveLinParamsHashCode * liPrime) + F_lrealToLintBits(stMcMoveParams.stMoveLinParams.lrVel);

METH_stMoveLinParamsHashCode := (METH_stMoveLinParamsHashCode * liPrime) + F_lrealToLintBits(stMcMoveParams.stMoveLinParams.lrAcc);

METH_stMoveLinParamsHashCode := (METH_stMoveLinParamsHashCode * liPrime) + F_lrealToLintBits(stMcMoveParams.stMoveLinParams.lrDec);

METH_stMoveLinParamsHashCode := (METH_stMoveLinParamsHashCode * liPrime) + F_lrealToLintBits(stMcMoveParams.stMoveLinParams.lrJrk);

METH_stMoveLinParamsHashCode := (METH_stMoveLinParamsHashCode * liPrime) + TO_LINT(stMcMoveParams.stMoveLinParams.smcCrdSys);

METH_stMoveLinParamsHashCode := (METH_stMoveLinParamsHashCode * liPrime) + TO_LINT(stMcMoveParams.stMoveLinParams.mcBufMode);

METH_stMoveLinParamsHashCode := (METH_stMoveLinParamsHashCode * liPrime) + TO_LINT(stMcMoveParams.stMoveLinParams.mcTrnMode);

FOR diIndx := LOWER_BOUND(stMcMoveParams.stMoveLinParams.arrTrnPrm, 1) TO UPPER_BOUND(stMcMoveParams.stMoveLinParams.arrTrnPrm, 1) BY 1 DO
  METH_stMoveLinParamsHashCode := (METH_stMoveLinParamsHashCode * liPrime) + F_lrealToLintBits(stMcMoveParams.stMoveLinParams.arrTrnPrm[diIndx]);
END_FOR

METH_stMoveLinParamsHashCode := (METH_stMoveLinParamsHashCode * liPrime) + TO_LINT(stMcMoveParams.stMoveLinParams.smcOrnMod);

METH_stMoveLinParamsHashCode := (METH_stMoveLinParamsHashCode * liPrime) + F_lrealToLintBits(stMcMoveParams.stMoveLinParams.lrVelFctr);

METH_stMoveLinParamsHashCode := (METH_stMoveLinParamsHashCode * liPrime) + F_lrealToLintBits(stMcMoveParams.stMoveLinParams.lrAccFctr);

METH_stMoveLinParamsHashCode := (METH_stMoveLinParamsHashCode * liPrime) + F_lrealToLintBits(stMcMoveParams.stMoveLinParams.lrJrkFctr);

                
END_METHOD

// based on https://stackoverflow.com/questions/113511/best-implementation-for-hashcode-method-for-a-collection/113600#113600
METHOD PRIVATE METH_mcMoveCrcRelHashCode : LINT
VAR_INPUT
  liPrime : LINT := 37;
END_VAR
VAR
  liInitVal : LINT := 1; // has to be nonzero
  diIndx    : DINT;
END_VAR
                  METH_mcMoveCrcRelHashCode := liInitVal;

METH_mcMoveCrcRelHashCode := (METH_mcMoveCrcRelHashCode * liPrime) + BOOL_TO_LINT(mcMoveCrcRel.Execute);

METH_mcMoveCrcRelHashCode := (METH_mcMoveCrcRelHashCode * liPrime) + TO_LINT(mcMoveCrcRel.CircMode);

FOR diIndx := LOWER_BOUND(mcMoveCrcRel.AuxPoint.v, 1) TO UPPER_BOUND(mcMoveCrcRel.AuxPoint.v, 1) BY 1 DO
  METH_mcMoveCrcRelHashCode := (METH_mcMoveCrcRelHashCode * liPrime) + F_lrealToLintBits(mcMoveCrcRel.AuxPoint.v[diIndx]);
END_FOR

FOR diIndx := LOWER_BOUND(mcMoveCrcRel.EndPoint.v, 1) TO UPPER_BOUND(mcMoveCrcRel.EndPoint.v, 1) BY 1 DO
  METH_mcMoveCrcRelHashCode := (METH_mcMoveCrcRelHashCode * liPrime) + F_lrealToLintBits(mcMoveCrcRel.EndPoint.v[diIndx]);
END_FOR

METH_mcMoveCrcRelHashCode := (METH_mcMoveCrcRelHashCode * liPrime) + TO_LINT(mcMoveCrcRel.PathChoice);

METH_mcMoveCrcRelHashCode := (METH_mcMoveCrcRelHashCode * liPrime) + F_lrealToLintBits(mcMoveCrcRel.Velocity);

METH_mcMoveCrcRelHashCode := (METH_mcMoveCrcRelHashCode * liPrime) + F_lrealToLintBits(mcMoveCrcRel.Acceleration);

METH_mcMoveCrcRelHashCode := (METH_mcMoveCrcRelHashCode * liPrime) + F_lrealToLintBits(mcMoveCrcRel.Deceleration);

METH_mcMoveCrcRelHashCode := (METH_mcMoveCrcRelHashCode * liPrime) + F_lrealToLintBits(mcMoveCrcRel.Jerk);

METH_mcMoveCrcRelHashCode := (METH_mcMoveCrcRelHashCode * liPrime) + TO_LINT(mcMoveCrcRel.CoordSystem);

METH_mcMoveCrcRelHashCode := (METH_mcMoveCrcRelHashCode * liPrime) + TO_LINT(mcMoveCrcRel.BufferMode);

METH_mcMoveCrcRelHashCode := (METH_mcMoveCrcRelHashCode * liPrime) + TO_LINT(mcMoveCrcRel.TransitionMode);

FOR diIndx := LOWER_BOUND(mcMoveCrcRel.TransitionParameter, 1) TO UPPER_BOUND(mcMoveCrcRel.TransitionParameter, 1) BY 1 DO
  METH_mcMoveCrcRelHashCode := (METH_mcMoveCrcRelHashCode * liPrime) + F_lrealToLintBits(mcMoveCrcRel.TransitionParameter[diIndx]);
END_FOR

METH_mcMoveCrcRelHashCode := (METH_mcMoveCrcRelHashCode * liPrime) + TO_LINT(mcMoveCrcRel.OrientationMode);

METH_mcMoveCrcRelHashCode := (METH_mcMoveCrcRelHashCode * liPrime) + F_lrealToLintBits(mcMoveCrcRel.VelFactor);

METH_mcMoveCrcRelHashCode := (METH_mcMoveCrcRelHashCode * liPrime) + F_lrealToLintBits(mcMoveCrcRel.AccFactor);

METH_mcMoveCrcRelHashCode := (METH_mcMoveCrcRelHashCode * liPrime) + F_lrealToLintBits(mcMoveCrcRel.JerkFactor);

                
END_METHOD

// based on https://stackoverflow.com/questions/113511/best-implementation-for-hashcode-method-for-a-collection/113600#113600
METHOD PRIVATE METH_mcMoveDirAbsHashCode : LINT
VAR_INPUT
  liPrime : LINT := 37;
END_VAR
VAR
  liInitVal : LINT := 1; // has to be nonzero
  diIndx    : DINT;
END_VAR
                  METH_mcMoveDirAbsHashCode := liInitVal;

METH_mcMoveDirAbsHashCode := (METH_mcMoveDirAbsHashCode * liPrime) + BOOL_TO_LINT(mcMoveDirAbs.Execute);

FOR diIndx := LOWER_BOUND(mcMoveDirAbs.Position.v, 1) TO UPPER_BOUND(mcMoveDirAbs.Position.v, 1) BY 1 DO
  METH_mcMoveDirAbsHashCode := (METH_mcMoveDirAbsHashCode * liPrime) + F_lrealToLintBits(mcMoveDirAbs.Position.v[diIndx]);
END_FOR

METH_mcMoveDirAbsHashCode := (METH_mcMoveDirAbsHashCode * liPrime) + TO_LINT(mcMoveDirAbs.MovementType);

METH_mcMoveDirAbsHashCode := (METH_mcMoveDirAbsHashCode * liPrime) + TO_LINT(mcMoveDirAbs.CoordSystem);

METH_mcMoveDirAbsHashCode := (METH_mcMoveDirAbsHashCode * liPrime) + TO_LINT(mcMoveDirAbs.BufferMode);

METH_mcMoveDirAbsHashCode := (METH_mcMoveDirAbsHashCode * liPrime) + TO_LINT(mcMoveDirAbs.TransitionMode);

FOR diIndx := LOWER_BOUND(mcMoveDirAbs.TransitionParameter, 1) TO UPPER_BOUND(mcMoveDirAbs.TransitionParameter, 1) BY 1 DO
  METH_mcMoveDirAbsHashCode := (METH_mcMoveDirAbsHashCode * liPrime) + F_lrealToLintBits(mcMoveDirAbs.TransitionParameter[diIndx]);
END_FOR

METH_mcMoveDirAbsHashCode := (METH_mcMoveDirAbsHashCode * liPrime) + F_lrealToLintBits(mcMoveDirAbs.VelFactor);

METH_mcMoveDirAbsHashCode := (METH_mcMoveDirAbsHashCode * liPrime) + F_lrealToLintBits(mcMoveDirAbs.AccFactor);

METH_mcMoveDirAbsHashCode := (METH_mcMoveDirAbsHashCode * liPrime) + F_lrealToLintBits(mcMoveDirAbs.JerkFactor);

                
END_METHOD

// based on https://stackoverflow.com/questions/113511/best-implementation-for-hashcode-method-for-a-collection/113600#113600
METHOD PRIVATE METH_mcMoveDirRelHashCode : LINT
VAR_INPUT
  liPrime : LINT := 37;
END_VAR
VAR
  liInitVal : LINT := 1; // has to be nonzero
  diIndx    : DINT;
END_VAR
                  METH_mcMoveDirRelHashCode := liInitVal;

METH_mcMoveDirRelHashCode := (METH_mcMoveDirRelHashCode * liPrime) + BOOL_TO_LINT(mcMoveDirRel.Execute);

FOR diIndx := LOWER_BOUND(mcMoveDirRel.Distance.v, 1) TO UPPER_BOUND(mcMoveDirRel.Distance.v, 1) BY 1 DO
  METH_mcMoveDirRelHashCode := (METH_mcMoveDirRelHashCode * liPrime) + F_lrealToLintBits(mcMoveDirRel.Distance.v[diIndx]);
END_FOR

METH_mcMoveDirRelHashCode := (METH_mcMoveDirRelHashCode * liPrime) + TO_LINT(mcMoveDirRel.MovementType);

METH_mcMoveDirRelHashCode := (METH_mcMoveDirRelHashCode * liPrime) + TO_LINT(mcMoveDirRel.CoordSystem);

METH_mcMoveDirRelHashCode := (METH_mcMoveDirRelHashCode * liPrime) + TO_LINT(mcMoveDirRel.BufferMode);

METH_mcMoveDirRelHashCode := (METH_mcMoveDirRelHashCode * liPrime) + TO_LINT(mcMoveDirRel.TransitionMode);

FOR diIndx := LOWER_BOUND(mcMoveDirRel.TransitionParameter, 1) TO UPPER_BOUND(mcMoveDirRel.TransitionParameter, 1) BY 1 DO
  METH_mcMoveDirRelHashCode := (METH_mcMoveDirRelHashCode * liPrime) + F_lrealToLintBits(mcMoveDirRel.TransitionParameter[diIndx]);
END_FOR

METH_mcMoveDirRelHashCode := (METH_mcMoveDirRelHashCode * liPrime) + F_lrealToLintBits(mcMoveDirRel.VelFactor);

METH_mcMoveDirRelHashCode := (METH_mcMoveDirRelHashCode * liPrime) + F_lrealToLintBits(mcMoveDirRel.AccFactor);

METH_mcMoveDirRelHashCode := (METH_mcMoveDirRelHashCode * liPrime) + F_lrealToLintBits(mcMoveDirRel.JerkFactor);

                
END_METHOD

// based on https://stackoverflow.com/questions/113511/best-implementation-for-hashcode-method-for-a-collection/113600#113600
METHOD PRIVATE METH_mcMoveLinAbsHashCode : LINT
VAR_INPUT
  liPrime : LINT := 37;
END_VAR
VAR
  liInitVal : LINT := 1; // has to be nonzero
  diIndx    : DINT;
END_VAR
                  METH_mcMoveLinAbsHashCode := liInitVal;

METH_mcMoveLinAbsHashCode := (METH_mcMoveLinAbsHashCode * liPrime) + BOOL_TO_LINT(mcMoveLinAbs.Execute);

FOR diIndx := LOWER_BOUND(mcMoveLinAbs.Position.v, 1) TO UPPER_BOUND(mcMoveLinAbs.Position.v, 1) BY 1 DO
  METH_mcMoveLinAbsHashCode := (METH_mcMoveLinAbsHashCode * liPrime) + F_lrealToLintBits(mcMoveLinAbs.Position.v[diIndx]);
END_FOR

METH_mcMoveLinAbsHashCode := (METH_mcMoveLinAbsHashCode * liPrime) + F_lrealToLintBits(mcMoveLinAbs.Velocity);

METH_mcMoveLinAbsHashCode := (METH_mcMoveLinAbsHashCode * liPrime) + F_lrealToLintBits(mcMoveLinAbs.Acceleration);

METH_mcMoveLinAbsHashCode := (METH_mcMoveLinAbsHashCode * liPrime) + F_lrealToLintBits(mcMoveLinAbs.Deceleration);

METH_mcMoveLinAbsHashCode := (METH_mcMoveLinAbsHashCode * liPrime) + F_lrealToLintBits(mcMoveLinAbs.Jerk);

METH_mcMoveLinAbsHashCode := (METH_mcMoveLinAbsHashCode * liPrime) + TO_LINT(mcMoveLinAbs.CoordSystem);

METH_mcMoveLinAbsHashCode := (METH_mcMoveLinAbsHashCode * liPrime) + TO_LINT(mcMoveLinAbs.BufferMode);

METH_mcMoveLinAbsHashCode := (METH_mcMoveLinAbsHashCode * liPrime) + TO_LINT(mcMoveLinAbs.TransitionMode);

FOR diIndx := LOWER_BOUND(mcMoveLinAbs.TransitionParameter, 1) TO UPPER_BOUND(mcMoveLinAbs.TransitionParameter, 1) BY 1 DO
  METH_mcMoveLinAbsHashCode := (METH_mcMoveLinAbsHashCode * liPrime) + F_lrealToLintBits(mcMoveLinAbs.TransitionParameter[diIndx]);
END_FOR

METH_mcMoveLinAbsHashCode := (METH_mcMoveLinAbsHashCode * liPrime) + TO_LINT(mcMoveLinAbs.OrientationMode);

METH_mcMoveLinAbsHashCode := (METH_mcMoveLinAbsHashCode * liPrime) + F_lrealToLintBits(mcMoveLinAbs.VelFactor);

METH_mcMoveLinAbsHashCode := (METH_mcMoveLinAbsHashCode * liPrime) + F_lrealToLintBits(mcMoveLinAbs.AccFactor);

METH_mcMoveLinAbsHashCode := (METH_mcMoveLinAbsHashCode * liPrime) + F_lrealToLintBits(mcMoveLinAbs.JerkFactor);

                
END_METHOD

// based on https://stackoverflow.com/questions/113511/best-implementation-for-hashcode-method-for-a-collection/113600#113600
METHOD PRIVATE METH_mcMoveLinRelHashCode : LINT
VAR_INPUT
  liPrime : LINT := 37;
END_VAR
VAR
  liInitVal : LINT := 1; // has to be nonzero
  diIndx    : DINT;
END_VAR
                  METH_mcMoveLinRelHashCode := liInitVal;

METH_mcMoveLinRelHashCode := (METH_mcMoveLinRelHashCode * liPrime) + BOOL_TO_LINT(mcMoveLinRel.Execute);

FOR diIndx := LOWER_BOUND(mcMoveLinRel.Distance.v, 1) TO UPPER_BOUND(mcMoveLinRel.Distance.v, 1) BY 1 DO
  METH_mcMoveLinRelHashCode := (METH_mcMoveLinRelHashCode * liPrime) + F_lrealToLintBits(mcMoveLinRel.Distance.v[diIndx]);
END_FOR

METH_mcMoveLinRelHashCode := (METH_mcMoveLinRelHashCode * liPrime) + F_lrealToLintBits(mcMoveLinRel.Velocity);

METH_mcMoveLinRelHashCode := (METH_mcMoveLinRelHashCode * liPrime) + F_lrealToLintBits(mcMoveLinRel.Acceleration);

METH_mcMoveLinRelHashCode := (METH_mcMoveLinRelHashCode * liPrime) + F_lrealToLintBits(mcMoveLinRel.Deceleration);

METH_mcMoveLinRelHashCode := (METH_mcMoveLinRelHashCode * liPrime) + F_lrealToLintBits(mcMoveLinRel.Jerk);

METH_mcMoveLinRelHashCode := (METH_mcMoveLinRelHashCode * liPrime) + TO_LINT(mcMoveLinRel.CoordSystem);

METH_mcMoveLinRelHashCode := (METH_mcMoveLinRelHashCode * liPrime) + TO_LINT(mcMoveLinRel.BufferMode);

METH_mcMoveLinRelHashCode := (METH_mcMoveLinRelHashCode * liPrime) + TO_LINT(mcMoveLinRel.TransitionMode);

FOR diIndx := LOWER_BOUND(mcMoveLinRel.TransitionParameter, 1) TO UPPER_BOUND(mcMoveLinRel.TransitionParameter, 1) BY 1 DO
  METH_mcMoveLinRelHashCode := (METH_mcMoveLinRelHashCode * liPrime) + F_lrealToLintBits(mcMoveLinRel.TransitionParameter[diIndx]);
END_FOR

METH_mcMoveLinRelHashCode := (METH_mcMoveLinRelHashCode * liPrime) + TO_LINT(mcMoveLinRel.OrientationMode);

METH_mcMoveLinRelHashCode := (METH_mcMoveLinRelHashCode * liPrime) + F_lrealToLintBits(mcMoveLinRel.VelFactor);

METH_mcMoveLinRelHashCode := (METH_mcMoveLinRelHashCode * liPrime) + F_lrealToLintBits(mcMoveLinRel.AccFactor);

METH_mcMoveLinRelHashCode := (METH_mcMoveLinRelHashCode * liPrime) + F_lrealToLintBits(mcMoveLinRel.JerkFactor);

                
END_METHOD

METHOD METH_executeMcMove
VAR_IN_OUT
  axisGrpRefSm3 : SM3_Robotics.AXIS_GROUP_REF_SM3;
END_VAR
VAR_OUTPUT
  xDone        : BOOL;
  xBusy        : BOOL;
  xActive      : BOOL;
  xCmdAborted  : BOOL;
  xCmdAccepted : BOOL;
  xError       : BOOL;
  smcError     : SM3_Error.SMC_ERROR;
  smcMvmtId    : SM3_Common.SMC_Movement_Id;
END_VAR
                  CASE stMcMoveParams.eMcMotionFbType OF

  E_mcMotionFbType.moveCrcAbs:
    fbLogAdd.METH_appendLog('Not implemented yet!', xNewline:=TRUE);

  E_mcMotionFbType.moveCrcRel:
    fbLogAdd.METH_appendLog('Not implemented yet!', xNewline:=TRUE);

  E_mcMotionFbType.moveDirAbs:
    mcMoveDirAbs(AxisGroup:=axisGrpRefSm3,
                 Execute:=TRUE,
                 Position:=stMcMoveParams.stMoveDirParams.smcPosRef,
                 MovementType:=stMcMoveParams.stMoveDirParams.smcPtpTyp,
                 CoordSystem:=stMcMoveParams.stMoveDirParams.smcCrdSys,
                 BufferMode:=stMcMoveParams.stMoveDirParams.mcBufMode,
                 TransitionMode:=stMcMoveParams.stMoveDirParams.mcTrnMode,
                 TransitionParameter:=stMcMoveParams.stMoveDirParams.arrTrnPrm,
                 VelFactor:=stMcMoveParams.stMoveDirParams.lrVelFctr,
                 AccFactor:=stMcMoveParams.stMoveDirParams.lrAccFctr,
                 JerkFactor:=stMcMoveParams.stMoveDirParams.lrJrkFctr,
                 Done=>xDone,
                 Busy=>xBusy,
                 Active=>xActive,
                 CommandAborted=>xCmdAborted,
                 CommandAccepted=>xCmdAccepted,
                 Error=>xError,
                 ErrorID=>smcError,
                 MovementId=>smcMvmtId);

  E_mcMotionFbType.moveDirRel:
    fbLogAdd.METH_appendLog('Not implemented yet!', xNewline:=TRUE);

  E_mcMotionFbType.moveLinAbs:
    fbLogAdd.METH_appendLog('Not implemented yet!', xNewline:=TRUE);

  E_mcMotionFbType.moveLinRel:
    fbLogAdd.METH_appendLog('Not implemented yet!', xNewline:=TRUE);

END_CASE

                
END_METHOD

METHOD METH_resetMcMove
VAR_IN_OUT
  axisGrpRefSm3 : SM3_Robotics.AXIS_GROUP_REF_SM3;
END_VAR
                  mcMoveDirAbs(AxisGroup:=axisGrpRefSm3,
             Execute:=FALSE);

                
END_METHOD

// IMPORTANT: Call UpdateElement() to ensure that the reference will be updated after an online change.
METHOD FB_reinit : BOOL
VAR_INPUT
END_VAR
                  UpdateElement(itfElement:=THIS^);

                
END_METHOD

